(* CODESYS project TcoCore.library
   Author: Inxton
   Placeholder: TcoCore
   Title: TcoCore
   Version: 0.4.2.453
   DefaultNamespace: TcoCore
   Company: Vortex.Library

Project tree, tasks and I/O mapping:
  libraries: Tc2_EtherCAT, * (Beckhoff Automation GmbH); Tc2_Standard, 3.3.3.0 (Beckhoff Automation GmbH); Tc2_System, 3.4.24.0 (Beckhoff Automation GmbH); Tc2_Utilities, 3.3.41.0 (Beckhoff Automation GmbH); Tc3_Module, 3.3.21.0 (Beckhoff Automation GmbH)
  DUTs/
  GVLs/
  POUs/
    Compatibility/
      function block TcoContextCompatibility [ST]: _Close, _Open
      function block TcoContextNfCompatibility [ST]: Main, VolatileClose, VolatileOpen
    Prototypes/
      TcoComponent/
        interface ITcoComponent
        interface ITcoServiceable: IsService, Service
        function block TcoComponent [ST]: CheckIfIsInServiceMode, FB_init, IsService, Restore, Service, ServiceMode
      TcoContext/
        interface ITcoContext: EndCycleCount, Environment, Rtc, StartCycleCount
        interface ITcoContextEnvironment: Messaging
        function block TcoContext [ST]: Close, Context, EndCycleCount, Environment, FB_init, Identity, Main, OnEntry, OnExit, Open, Rtc, RtcSynchronize, Run, StartCycleCount
        function block TcoContextEnvironment [ST]: Messaging
      TcoMessage/
        data type eMessageCategory
        interface ITcoMessenger: Debug, Error, Info, Notify, Post, Programming, Trace, Warning
        interface ITcoMessengerSettings: IsSuspended, MinLevel, Resume, Suspend
        data type TcoMessage
        function block TcoMessenger [ST]: Catastrophic, Critical, Debug, Error, Info, Notify, Programming, Trace, Warning, Clear, Compose, FB_init, Post
        function block TcoMessengerSettings [ST]: IsSuspended, MinLevel, Resume, Suspend
      TcoObject/
        interface ITcoObject: Context, Identity
        function block TcoObject [ST]: Context, EqualsTo, FB_init, Identity, Messenger
      TcoRestorable/
        interface ITcoObjectRestorer: RestoreObject
        interface ITcoRestorable: Restore
      TcoRtc/
        interface ITcoRtc: IsSynchronized, IsValid, NowLocal, NowLocalAsTIMESTRUCT, NowUTC, NowUTCAsTIMESTRUCT, TickClock
        program RtcPrg [ST]: Synchronize
        data type RtcSynchParams
        function block TcoRtc [ST]: IsSynchronized, IsValid, NowLocal, NowLocalAsTIMESTRUCT, NowUTC, NowUTCAsTIMESTRUCT, TickClock, Update
      TcoSequencer/
        data type eSequencerError
        data type eSequencerMode
        data type eStepStatus
        interface ITcoSequencer: CurrentStep, ModeController, Run
        interface ITcoSequencerModeController: Mode, StepBackward, StepForward, StepIn
        data type StepDetails
        function block TcoSequencer [ST]: CheckStepId, Close, CompleteSequence, CompleteStep, CurrentStep, FB_init, IsStepIdUnique, Main, ModeController, OnlineChange, OnSequenceCompleted, OnSequencerError, OnStepCompleted, Open, RequestStep, Restore, Run, Step, StepChanged, StepCompleteWhen, StepInternal
        function block TcoSequencerModeController [ST]: ChangeMode, DisableModeChanging, DisableStepSkipping, Mode, OnModeChange, StepBackward, StepForward, StepIn
      TcoState/
        data type eRestoreMode
        interface ITcoState: IsAutoRestoreEnabled, LastStateChangeCycle, RestoreObject, State
        function block TcoState [ST]: ChangeState
        function block TcoStateBase [ST]: AutoRestorable, AutoRestore, ChangeStateProtected, CheckIfAutoRestoreEnabledByParent, CheckIfCalledCyclically, Context, FB_init, Identity, IsAutoRestoreEnabled, LastStateChangeCycle, OnStateChange, Restore, RestoreObject, State
        function block TcoStateExtendible [ST]: ChangeState
      TcoTask/
        data type eTaskState
        interface ITcoTask: Abort, Busy, Done, Error, Invoke
        interface ITcoTaskStatus: Busy, Done, Error
        function block TcoTask [ST]: Abort, AutoRestorable, AutoRestore, Busy, CheckIfAutoRestoreEnabledByParent, CheckIfCalledCyclically, Context, Done, DoneWhen, ElapsedTime, Enabled, Error, Execute, FB_init, Identity, Invoke, OnAbort, OnDone, OnTaskError, Ready, Restore, State, ThrowWhen
    TestFixtures/
      function block _internals_TcoContext [ST]: _Close, _GetSynchParams, _Open, _rtcUpdate, ProbeRun
      function block _internals_TcoSequencer [ST]: _Close, _Open
    Utilities/
      function block StringBuilder [ST]: Append, Clear, ToString
    program MAIN [ST]
*)

// POUs/Prototypes/TcoMessage/eMessageCategory
(*~
	<docu>
		<summary>
			Message categories.
		</summary>
	</docu>	
~*)

// ATTENTION: Values must be multiply of 100
{attribute 'qualified_only'}
{attribute 'strict'}
TYPE eMessageCategory :
(		
	All := 0,
	(*~
	<docu>
		<summary>
			Debug message to be used for debugging purpose only.
			Use when you need to report debug information for you as programmer. 
		</summary>
	</docu>	
	~*)	
	Debug := 100,
	(*~
	<docu>
		<summary>
			Trace message to be used for tracing purpose.
			Use when you need to track detailed information about internal states of the program for detailed visibility. 
			This is lowest level of category that can be used in production, for detailed observation of PLC program.
		</summary>
	</docu>	
	~*)	
	Trace := 200,
	(*~
	<docu>
		<summary>
			Info message.
			Use when you want to deliver information to the user, that has only informative character and does not adversely affect a process.
		</summary>
	</docu>	
	~*)	
	Info := 300,
	(*~
	<docu>
		<summary>
			Time-out message.
			Use this category when you want to report a timed-out information, that may eventually succed.
		</summary>
	</docu>	
	~*)
	TimedOut := 400,
	(*~
	<docu>
		<summary>
			Notification message.
			Use this category when you want to report a notification that may be of interest to the user, but does not adversly affect a process.
		</summary>
	</docu>	
	~*)
	Notification := 500,
	(*~
	<docu>
		<summary>
			Warning message.
			Use this category when you want to report to the user an information about a possible problem, that may adversly affect a process.
			Information in this cateogory aims to help the user to identify a problem, the cause of such problem does not necessarily stops the process.
		</summary>
	</docu>	
	~*)
	Warning := 600,
	(*~
	<docu>
		<summary>
			Error message.
			Use this categoty when there is a failure that cannot be immediately recovered and an intervention is needed. This is typically a situation when a device fails
			to deliver expected result. 
			Do not use this category to report information about failed process like measurement or detection.
		</summary>
	</docu>	
	~*)
	Error := 700,	
	(*~
	<docu>
		<summary>
			Programming issue.
			Use this category to inform about a possible programming error, defect in settings or missing information at a level of programming or system or process settings. 
		</summary>
	</docu>	
	~*)
	ProgrammingError := 900,
	(*~
	<docu>
		<summary>
			Critical error. 
			Use this category when a critical error occured, that is not recoverable by the means of software (reset/restore) and a detailed inspection is required.
		</summary>
	</docu>	
	~*)	
	Critical := 1000,		
	(*~
	<docu>
		<summary>
			Catastrophic error. 
			Use this category when there is a situation when the device cannot continue operations due to irrecoverable failure.
		</summary>
	</docu>	
	~*)
	Catastrophic := 1100,
	
	None := 32767
);
END_TYPE

// POUs/Prototypes/TcoMessage/TcoMessage
(*~
	<docu>
		<summary>
			Complete message details including time stamp, message text, message category, identity of the message provider, context cycle in which the message was posted.			
		</summary>				
	</docu>	
~*)
TYPE TcoMessage :
STRUCT
(*~
	<docu>
		<summary>
			Time when the message was posted.
		</summary>				
	</docu>	
~*)
	{attribute clr [ReadOnly()]}
	TimeStamp : DT;
(*~
	<docu>
		<summary>
			Text of the message.
		</summary>				
	</docu>	
~*)
	{attribute clr [ReadOnly()]}		
	Text : STRING(125);
(*~
	<docu>
		<summary>
			Identity of the TcoObject that posted this message. 
		</summary>				
	</docu>	
~*)
	{attribute clr [ReadOnly()]}	
	Identity : ULINT;	
(*~
	<docu>
		<summary>
			Message category of this message. See <see cref="eMessageCategory"/> for detailed informations. 
		</summary>				
	</docu>	
~*)
	Category : eMessageCategory;
(*~
	<docu>
		<summary>
			Context cycle in which the message was posted.
		</summary>				
	</docu>	
~*)
	{attribute clr [ReadOnly()]}
	Cycle : ULINT;
	
(*~
	<docu>
		<summary>
			Count of messages of the object in the current cycle.
		</summary>				
	</docu>	
~*)
	{attribute clr [ReadOnly()]}
	PerCycleCount : BYTE;
END_STRUCT
END_TYPE

// POUs/Prototypes/TcoRtc/RtcSynchParams
TYPE RtcSynchParams :
STRUCT
	synchContextIdentity	:	ULINT;
	doSynch					:	BOOL;
	syncAmsId				:	STRING;
	syncPeriod				:	UINT; 
END_STRUCT
END_TYPE

// POUs/Prototypes/TcoSequencer/eSequencerError
(*~
	<docu>
		<summary>
			Describes cause of the sequencer error.
		</summary>				
	</docu>	
~*)
{attribute 'qualified_only'}
{attribute 'strict'}
TYPE eSequencerError :
(
(*~
	<docu>
		<summary>
			No error.
		</summary>				
	</docu>	
~*)	
	noError := 0,
(*~
	<docu>
		<summary>
			Some of the StepId in the sequence is not unique (```TcoSequencer.Step(StepID)```).
		</summary>				
	</docu>	
~*)	
	NotUniqueStepId := 10,
(*~
	<docu>
		<summary>
			StepId of the currently executed step has been changed during execution.
		</summary>				
	</docu>	
~*)
	StepIdHasBeenChanged := 20,
(*~
	<docu>
		<summary>
			Order of the currently executed step has been changed during execution.
		</summary>				
	</docu>	
~*)
	OrderOfTheStepHasBeenChanged := 40,
(*~
	<docu>
		<summary>
			Method ```RequestStep``` has been called with nonexisting StepId.
		</summary>				
	</docu>	
~*)
	StepWithRequestedIdDoesNotExists := 50,
(*~
	<docu>
		<summary>
			Multiple simultaneous calls of ```RequestStep()```. Another ```RequestStep()``` method has been called while previous ```RequestStep()``` call has not yet been completed.
		</summary>				
	</docu>	
~*)
	MultipleRequestStepMethodCall := 60,
(*~
	<docu>
		<summary>
			StepId is bellow min. range. Minimal value is -32767.
		</summary>				
	</docu>	
~*)
	StepIdTooLow := 70,
(*~
	<docu>
		<summary>
			StepId is above max range. Maximal value is 32766.
		</summary>				
	</docu>	
~*)
	StepIdTooHigh := 80,
(*~
	<docu>
		<summary>
			Mode of the sequencer is invalid.
		</summary>				
	</docu>	
~*)
	InvalidSequencerMode := 90
);
END_TYPE

// POUs/Prototypes/TcoSequencer/eSequencerMode
(*~
	<docu>
		<summary>
			Modes of the sequencer.
		</summary>				
	</docu>	
~*)	
{attribute 'qualified_only'}
{attribute 'strict'}
TYPE eSequencerMode :
(
(*~
	<docu>
		<summary>
			Invalid, no logic is executed.
		</summary>				
	</docu>	
~*)	
	Invalid := -10,
(*~
	<docu>
		<summary>
			Sequencer runs the steps of the sequence. 
			(When cyclic mode is selected, next step is automatically started after the previous one has been completed.)
		</summary>				
	</docu>	
~*)	
	CyclicMode := 0,
(*~
	<docu>
		<summary>
		    Sequencer is in mode of step-by-step operation. The current step completes the execution regularly.
			In this mode the Step Forward/Backward and manual step execution is available.			
			<para>
				See <see cref="TcoSequencerModeController.PlcTcoSequencerModeController.StepForward()"/> for detailed description.
				See <see cref="TcoSequencerModeController.PlcTcoSequencerModeController.StepIn()"/> for detailed description.
				See <see cref="TcoSequencerModeController.PlcTcoSequencerModeController.StepBackward()"/> for detailed description.
			</para>
		</summary>				
	</docu>	
~*)	
	StepMode := 10
);
END_TYPE

// POUs/Prototypes/TcoSequencer/eStepStatus
(*~
	<docu>
		<summary>
			Describes the step status inside the sequencer.
		</summary>				
	</docu>	
~*)
{attribute 'qualified_only'}
{attribute 'strict'}
TYPE eStepStatus :
(
(*~
	<docu>
		<summary>
			No status defined.
		</summary>				
	</docu>	
~*)	
	None := 0,
(*~
	<docu>
		<summary>
			Step is disabled and won't be executed.
			Next enabled step in the sequence will be executed, when the sequencer reaches that step.
		</summary>				
	</docu>	
~*)	
	Disabled := 10,
(*~
	<docu>
		<summary>
			Step is ready to run. This case occurs when sequence is in step mode, step is in order of the execution and step is enabled.
			The body statements of the current step's are not executing. After calling StepIn method, step starts running the statements.
		</summary>				
	</docu>	
~*)	
	ReadyToRun := 20,
(*~
	<docu>
		<summary>
			Step is currently running (The body statements are running).
		</summary>				
	</docu>	
~*)	
	Running := 30,	
(*~
	<docu>
		<summary>
			Step has finished (The body statements are not running).
		</summary>				
	</docu>	
~*)	
	Done := 40,
(*~
	<docu>
		<summary>
			Step is in error state. The sequencer does not execute any step logic.
		</summary>				
	</docu>	
~*)	
	Error := 50
);
END_TYPE

// POUs/Prototypes/TcoSequencer/StepDetails
(*~
	<docu>
		<summary>
			Describes the status of a step of the sequencer.
		</summary>				
	</docu>	
~*)
TYPE StepDetails :
STRUCT
(*~
	<docu>
		<summary>
			Step identification number.
		</summary>	
		<remarks>			
 			<note type="important">
				This number must be unique throughout the complete sequence. It is required to uniquely identify the step of the sequence.
			</note>
			<para>
				The <see cref="TcoSequencer.PlcTcoSequencer.RequestStep"/> method is using this number to jump to the required step.
			</para>
		</remarks>
	</docu>	
~*)
	{attribute addProperty Name "<#Step ID#>"}
	ID: INT;
(*~
	<docu>
		<summary>
			Order of the step in the sequence.
		</summary>	
	</docu>	
~*)
	{attribute addProperty Name "<#Step Order#>"}
	Order: UINT;
(*~
	<docu>
		<summary>
			If this value is false, step body is not executed and execution is moved to the next enabled step in the sequence.
		</summary>				
	</docu>	
~*)
	{attribute addProperty Name "<#Enabled#>"}
	Enabled: BOOL;
(*~
	<docu>
		<summary>
			Step description text.
		</summary>				
	</docu>	
~*)
	{attribute addProperty Name "<#Step description#>"}
	Description: STRING(254);
(*~
	<docu>
		<summary>
			Describes step status.
		</summary>				
		<remarks>			
			<para>
				See <see cref="eStepStatus"/> for detailed description.
			</para>
		</remarks>		
		enumStepStatus
	</docu>	
~*)	
	{attribute addProperty Name "<#Step status#>"}
	Status : eStepStatus;
(*~
	<docu>
		<summary>
			Step duration time.
		</summary>				
	</docu>	
~*)	
	{attribute addProperty Name "<#Step duration#>"}
	Duration : TIME;
END_STRUCT
END_TYPE

// POUs/Prototypes/TcoState/eRestoreMode
{attribute 'qualified_only'}
{attribute 'strict'}
TYPE eRestoreMode :
(
	None := 0,
	
	(*~
	<docu>
		<summary>
				Activates automatic restore mechanism for all immediate children (direct members).
		</summary>				
	</docu>	
	~*)	
	AutoRestoreMembers := 10
);
END_TYPE

// POUs/Prototypes/TcoTask/eTaskState
(*~
	<docu>
		<summary>
			Describes the state of the respective task.
		</summary>				
	</docu>	
~*)
{attribute 'qualified_only'}
{attribute 'strict'}
TYPE eTaskState :
(
(*~
	<docu>
		<summary>
			Task is in Ready state, the Execute() method returns FALSE. 
			Task can be started by calling the Invoke() method. 
		</summary>				
	</docu>	
~*)
	Ready := 0,
(*~
	<docu>
		<summary>
			Task is in Requested state, if Invoke() method has been called and the Execute() method has not been called yet. The first following call of the method Execute() 
			change the task state to Executing and returns TRUE, until Done or Error state is reached.
		</summary>				
	</docu>	
~*)
	Requested := 10,
(*~
	<docu>
		<summary>
			When the task is in Busy state, Execute() method returns TRUE. Leaving this state is possible as follows:
			<para>1.) By calling the Abort() task gets into the Idle state.</para>
			<para>2.) By calling the DoneWhen(true) task gets into the Done state.</para>
			<para>3.) By calling the Restore() task gets into the Idle state.</para>
			<para>4.) By calling the ThrowWhen(true) task gets into the Error state.</para>
		</summary>				
	</docu>	
~*)
	Busy := 20,
(*~
	<docu>
		<summary>
			Task is in Error state. To be able to start the task again the error state has to be reseted by calling the Restore() method.
		</summary>				
	</docu>	
~*)	
	Error := 30,
(*~
	<docu>
		<summary>
			Task is in Done state, Execute() method returns FALSE. To be able to start the task again '''rising edge''' of the calling of the Invoke() method needs to be performed.
			<p>Analogously to the xExecute signal of the <a href="https://plcopen.org/sites/default/files/downloads/creating_plcopen_compliant_function_block_libraries.pdf" title="Title"> PLCopen </a> motion function blocks.</p>
		</summary>				
	</docu>	
~*)	
	Done := 40
);
END_TYPE

// POUs/Compatibility/TcoContextCompatibility
{attribute 'hide'}
{attribute clr [ExcludeFromApiDocumentation()]}
FUNCTION_BLOCK ABSTRACT TcoContextCompatibility EXTENDS TcoContext

{attribute 'hide'}
METHOD PROTECTED FINAL _Close
THIS^.Close();
END_METHOD

{attribute 'hide'}
METHOD PROTECTED FINAL _Open
THIS^.Open();
END_METHOD

END_FUNCTION_BLOCK

// POUs/Prototypes/TcoContext/TcoContext

(*~
	<docu>
		<summary>
			Root construction container, provides context information for <c>TcoObjects</c> declared within its scope.
			This function block is ```abstract``` and cannot be instantiated. 
			Use <see cref="TcoContext.PlcTcoContext.Run()"/> to run this context, ```Run``` method must be called only once per PLC Task cycle.
			Several 'TcoContext' instances can be declared and called inside one TwinCAT PlcTask, but only once per PLC cycle. 
			The instance should not be accessed from several Twincat PlcTasks.
			Default implemenation of the 'TcoContext' allows its child members access properties <see cref="TcoContext.PlcTcoContext.StartCycleCount()"/> 
			and <see cref="TcoContext.PlcTcoContext.EndCycleCount()"/>, messenger settings, rtc and other information related to the context of the running logic.			 			 			
			<note type="tip">
				 A <c>TcoContext</c> can contain objects, components and PLC logic of one independent station of the machine, 
				 while the another one can cover the same for another station.			
			</note>
			<remarks>			
				<note type="tip">
					TwinCAT PlcTask and <see cref="TcoTask.PlcTcoTask()"/> refer to two different concepts. 
				</note>
			</remarks>
		</summary>	
		<example>
			Declaration part of the 'TcoContext' example. 
		</example>
		<example>
				[!code-pas[Main](~/../TcOpen/src/TcoApplicationExamples/XaeAppExamples/PlcAppExamples/POUs/Context/VitoCorleone_Context.TcPOU?name=ContextExampleDeclarations)]
		</example>
		<example>
			Implementation part of the 'TcoContext' example.
		</example>
		<example>
				[!code-pas[Main](~/../TcOpen/src/TcoApplicationExamples/XaeAppExamples/PlcAppExamples/POUs/Context/VitoCorleone_Context.TcPOU?name=ContextExampleCode)]
		</example>
	</docu>	
~*)
FUNCTION_BLOCK PUBLIC ABSTRACT TcoContext IMPLEMENTS ITcoContext
VAR
	(*~
		<docu>
			<summary>
				Identity of this <c>TcoContext</c>.
				This variable is used in the higher level applications, 
				it allows to identify the context in SCADA like applications.	  
			</summary>			
		</docu>	
	~*)
	{attribute clr [RenderIgnore()]}
	{attribute clr [ReadOnly()]}
	_Identity : ULINT;
	{attribute clr [ReadOnly()]}
	_startCycleCount : ULINT;
	{attribute clr [ReadOnly()]}
	_endCycleCount : ULINT;
	_messagingLevel : eMessageCategory;
	{attribute clr [ReadOnly()]}
	_rtc : TcoRtc;
	{attribute clr [RenderIgnore()]}
    _settings : TcoContextEnvironment;	
END_VAR

(*~
	<docu>
		<summary>
			This method is called implicitly at the entry point of this context (<see cref="TcoContext.PlcTcoContext.Run()"/>).
			<remarks>			
				<note type="important">
					Do not call this method explicitly!
				</note>
			</remarks>
		</summary>			
	</docu>	
~*)
METHOD INTERNAL FINAL Close
_endCycleCount := _startCycleCount;
END_METHOD

(*~
	<docu>
		<summary>
			Returns reference to this instance of the <see cref="TcoContext.PlcTcoContext()"/>.
		</summary>			
	</docu>	
~*)
PROPERTY Context : ITcoContext
GET
Context := THIS^;
END_GET
END_PROPERTY

(*~
	<docu>
		<summary>
		    Gets the value of the counter incrememented by '1' at the end of each execution of this <see cref="TcoContext.PlcTcoContext()"/>.			
		</summary>			
	</docu>	
~*)
PROPERTY EndCycleCount : ULINT
GET
EndCycleCount := _endCycleCount;
END_GET
END_PROPERTY

PROPERTY Environment : ITcoContextEnvironment
GET
Environment := _settings;
END_GET
END_PROPERTY

METHOD FB_init : BOOL
VAR_INPUT
	bInitRetains : BOOL; // if TRUE, the retain variables are initialized (warm start / cold start)
	bInCopyCode : BOOL;  // if TRUE, the instance afterwards gets moved into the copy code (online change)
END_VAR
_Identity := ADR(THIS^);
END_METHOD

(*~
	<docu>
		<summary>
			Returns the identity of this <see cref ="TcoContext.PlcTcoContext()"/>. 
			This value is assigned when instantiated and cannot be changed at runtime.
			This member is used in the higher level applications.  
		</summary>			
	</docu>	
~*)
PROPERTY Identity : ULINT
GET
Identity := _Identity;
END_GET
END_PROPERTY

(*~
	<docu>
		<summary>
			Main method of the TcoContext. This is the entry point of any control logic that belongs to this context. 
			The call of this method is ensured by calling the <c>InstanceName.Run()</c> method, and it must not be called explicitly.
			This method is abstract, and it must be overridden in derived block.
		</summary>
	</docu>
~*)
METHOD PROTECTED ABSTRACT Main
END_METHOD

(*~
	<docu>
		<summary>
			Called on entry into context. When overridden in derived class allows to execute an arbitrary logic prior to opening the context cycle.
			<remarks>			
				<note type="important">					
					The method executes prior to opening the context. The context might not be properly initialized on first call. 
					Any information contained in the context at this point are from the last execution.
				</note>
			</remarks>
		</summary>			
	</docu>	
~*)
METHOD PROTECTED OnEntry
END_METHOD


(*~
	<docu>
		<summary>
			Called upon exit from the context. When overridden in derived class allows to execute an arbitrary logic after closing the context cycle.	
		</summary>			
	</docu>	
~*)METHOD PROTECTED OnExit
END_METHOD

(*~
	<docu>
		<summary>
			This method is called implicitly at the entry point of this context (<see cref="TcoContext.PlcTcoContext.Run()"/>).
			<remarks>			
				<note type="important">
					Do not call this method explicitly.
				</note>
			</remarks>
		</summary>			
	</docu>	
~*)
METHOD INTERNAL FINAL Open
_startCycleCount := _startCycleCount + 1;
_rtc.Update();
END_METHOD

PROPERTY Rtc : ITcoRtc
GET
Rtc := _rtc;
END_GET
END_PROPERTY

(*~
	<docu>
		<summary>
			Syncronizes the Real Time Clock (RTC) from given source.
			<remarks>			
				<note type="important">
					There is single RTC source for entire application. All context share the same RTC source.
				</note>
			</remarks>
		</summary>			
	</docu>	
~*)
METHOD RtcSynchronize  : REFERENCE TO TcoContext
VAR_INPUT
	(*~
		<docu>
			<summary>
				When called with true the synchronization mechanism executes.		
			</summary>			
		</docu>	
	~*)
	inDoSynch				:	BOOL;
	(*~
		<docu>
			<summary>
				```AMS ID``` of the system against which RTC of this application will synchronize.			
			</summary>			
		</docu>	
	~*)
	inSyncAmsId				:	STRING;
	(*~
		<docu>
			<summary>
				Set the synchronisation period.		
			</summary>			
		</docu>	
	~*)
	inSyncPeriod			:	UINT; 
END_VAR

VAR
	_RtcSynchParams			:	RtcSynchParams;			
END_VAR
_RtcSynchParams.doSynch					:=	inDoSynch;
_RtcSynchParams.syncAmsId				:=	inSyncAmsId;
_RtcSynchParams.syncPeriod				:=	inSyncPeriod;
_RtcSynchParams.synchContextIdentity	:=	THIS^._Identity;
RtcPrg.Synchronize(_RtcSynchParams);
RtcSynchronize REF= THIS^;
END_METHOD

(*~
	<docu>
		<summary>
			<para>
				This method executes of this context. It provided correct order of execution order of inner methods. Any logic of this context must be called within <see cref="TcoContext.PlcTcoContext.Main()"/>
				method. This method is final, so it cannot be overriden. The <c>InstanceName.Run()</c> needs to be called cyclically.
			</para>
		</summary>			
	</docu>	
~*)
METHOD PUBLIC FINAL Run
THIS^.OnEntry();
THIS^.Open();
THIS^.Main();
THIS^.Close();
THIS^.OnExit();
END_METHOD

(*~
	<docu>
		<summary>
		    Gets number of executions of this context. Value of this property is incremented by '1' at the beginning of the <see cref="TcoContext.PlcTcoContext()"/>. 			 			
		</summary>			
	</docu>	
~*)
PROPERTY StartCycleCount : ULINT
GET
StartCycleCount := _startCycleCount;
END_GET
END_PROPERTY

END_FUNCTION_BLOCK

// POUs/Prototypes/TcoTask/TcoTask
(*~
	<docu>
		<summary>
			Provides basic task execution. Task could be started by calling the <see cref="TcoTask.PlcTcoTask.Invoke()"/> method. The  <see cref="TcoTask.PlcTcoTask.Execute()"/> method returns true, until the task reaches the Done state.
			<para>
				To get the actual state of the task, <see cref="TcoTask.PlcTcoTask.Ready()"/>, <see cref="TcoTask.PlcTcoTask.Busy()"/>, <see cref="TcoTask.PlcTcoTask.Error()"/> and <see cref="TcoTask.PlcTcoTask.Done()"/> properties are available.
			</para>
		</summary>
		<example>
			Declaration part of the 'TcoTask' example. 
		</example>
		<example>
			[!code-pas[Main](~/../TcOpen/src/TcoApplicationExamples/XaeAppExamples/PlcAppExamples/POUs/Task/AskForTheFavor_Task.TcPOU?name=TaskExampleDeclarations)]
		</example>
		<example>
			Implementation part of the 'TcoTask' example.
		</example>
		<example>
			[!code-pas[Main](~/../TcOpen/src/TcoApplicationExamples/XaeAppExamples/PlcAppExamples/POUs/Task/AskForTheFavor_Task.TcPOU?name=TaskBodyExampleCode)]
		</example>
		<example>
			Example of the invoking this example 'TcoTask' instance 'outside' of the instance and wait if it ends-up in 'DONE' state or in 'ERROR' state.
		</example>
		<example>
			[!code-pas[Main](~/../TcOpen/src/TcoApplicationExamples/XaeAppExamples/PlcAppExamples/POUs/Sequencer/MakeAnOfferThatCantBeRefused.TcPOU?name=TaskExternalUseExample)]
		</example>
	</docu>	
~*)	
FUNCTION_BLOCK TcoTask EXTENDS TcoObject IMPLEMENTS ITcoTask, ITcoTaskStatus
VAR
	{attribute clr [ReadOnly()]}
	_taskState : eTaskState;
	{attribute 'hide'}
	_nextExpectedCycle : ULINT;
	{attribute 'hide'}
	_AutoRestorable : BOOL;
	{attribute 'hide'}
	_StartCycleCount	: ULINT;
	{attribute 'hide'}
	_MyParentsChangeStateCycle	: ULINT;
	{attribute 'hide'}
	_MyParentsLastChangeState	: INT;	
(*~
	<docu>
		<summary>
			Use to restore this instance to the Ready state. The value is than set to FALSE.			
		</summary>		
	</docu>	
~*)	
	{attribute addProperty Name "<#Restore request#>"}
	_restoreRequest : BOOL;
(*~
	<docu>
		<summary>
			Use to start the execution of the task from Ready state or from Done state by performing the rising edge. 
			<p>Analogously to the xExecute signal of the <a href="https://plcopen.org/sites/default/files/downloads/creating_plcopen_compliant_function_block_libraries.pdf" title="Title"> PLCopen </a> motion function blocks.</p>			
		</summary>			
	</docu>	
~*)
	{attribute addProperty Name "<#Invoke request#>"}
	_invokeRequest : BOOL;
(*~
	<docu>
		<summary>
			Use to abort the executing task and set this instance back to the Ready state.
			The value is than set to FALSE. 
		</summary>			
	</docu>	
~*)
	{attribute addProperty Name "<#Abort request#>"}
	_abortRequest : BOOL;	
(*~
	<docu>
		<summary>
			Use to determine if the task execution is enabled for example from the HMI application. 
			This value is read only, to modify it use the property <see cref="TcoTask.PlcTcoTask.Enabled()"/>		
		</summary>		
	</docu>	
~*)	
	{attribute addProperty Name "<#Enabled#>"}
	{attribute clr [ReadOnly()]}
	_enabled : BOOL := TRUE;
END_VAR

VAR	
	{attribute 'hide'}
	_executionTimer : Tc2_Standard.TON;
	{attribute clr [ReadOnly()]}
	_elapsedTime : TIME;
END_VAR

(*~
	<docu>
		<summary>
			Aborts the execution of this task and restores the ready state.			
		</summary>			
	</docu>	
~*)
METHOD Abort
IF THIS^._taskState = eTaskState.Busy THEN
	OnAbort();
	THIS^.Restore();
END_IF
END_METHOD

(*~
	<docu>
		<summary>
			Gets whether this instance is auto restorable. This is depends on the parent's settings; the value of this property is given by the parent of this object. 
			This value is assigned after download by calling the implicit method <c>FB_init()</c> of the parent object and cannot be changed during runtime.
			The <c>AutoRestorable</c> property of this objects is retrieved from the <c>EnableAutoRestore</c> property of the parent object.
			This is done by calling the <c>CheckIfAutoRestoreEnabledByParent()</c> method inside the implicit method <c>FB_init()</c> after download.
			If this instance is the auto restorable it will call the <see cref="TcoTask.PlcTcoTask.Restore()"/> method if:
			<para>
				1.) The <see cref="TcoTask.PlcTcoTask.Invoke()"/> method has not been called for one or more cycles and starts to be called again.
			</para>
			<para>
				2.)	Parent object of this instance changes its state.
			</para>
			<para>
				See also <see cref="TcoTask.PlcTcoTask.EnableAutoRestore()"/>
			</para>
		</summary>			
	</docu>	
~*)
PROPERTY AutoRestorable : BOOL
GET
AutoRestorable := _AutoRestorable;
END_GET
END_PROPERTY

(*~
	<docu>
		<summary>
			Private method called each time that the <see cref="TcoTask.PlcTcoTask.Execute()"/> method is called. If this instance is auto restorable, this method ensures calling the <see cref="TcoTask.PlcTcoTask.Restore()"/> method if:
			<para>
				1.)	Parent object of this instance changes its state in this Plc cycle.
			</para>
			<para>
				2.)	Parent object of this instance changes its state no mather when and this instance has not yet process this change.
			</para>
			<para>
				3.) The <see cref="TcoTask.PlcTcoTask.Invoke()"/> method has not been called for one or more cycles and starts to be called again.
			</para>
			<para>
				See also <see cref="TcoTask.PlcTcoTask.AutoRestorable()"/>
			</para>
			<para>
				See also <see cref="TcoTask.PlcTcoTask.EnableAutoRestore()"/>
			</para>
		</summary>			
	</docu>	
~*)
METHOD PRIVATE AutoRestore
VAR 
	_MyParent_TcoState	: ITcoState := 0;
	_MyParent_ChangeStateCycle : ULINT;
	_MyParent_LastChangeState : INT;
END_VAR
// If the parent of this instance is TcoState type or its derived type and the parent
// EnableAutoRestore property is set to TRUE, this instance determines the value
// of its own AutoRestorable property by calling CheckIfAutoRestoreEnabledByParent 
// after each download.
IF _AutoRestorable THEN		
	IF __QUERYINTERFACE(THIS^._Parent,_MyParent_TcoState) THEN 
		_MyParent_ChangeStateCycle := _MyParent_TcoState.LastStateChangeCycle;
		_MyParent_LastChangeState := _MyParent_TcoState.State;
	END_IF;	
	//If OnStateChange event of the parent has occured, the value of the parent's 
	//StartCycleCount property is stored into its ChangeStateCycle property.
	//Each child has to deal with it individually in the next call of its body,
	//restore itself, and copy the parent's ChangeStateCycle property into the
	//child's own property.
	IF _MyParent_ChangeStateCycle <> _MyParentsChangeStateCycle THEN
		Restore();
		_MyParentsChangeStateCycle := _MyParent_ChangeStateCycle;
	END_IF
	IF _MyParent_LastChangeState <> _MyParentsLastChangeState THEN
		Restore();
		_MyParentsLastChangeState := _MyParent_LastChangeState;
	END_IF
END_IF
END_METHOD

(*~
	<docu>
		<summary>
			Gets whether the task is executing.
		</summary>			
	</docu>	
~*)
PROPERTY Busy : BOOL
GET
Busy := THIS^._taskState = eTaskState.Busy;
END_GET
END_PROPERTY

(*~
	<docu>
		<summary>
			This method ensures reading out the parent's <see cref="TcoState.PlcTcoState.EnableAutoRestore()/> property and writing it into the <see cref="TcoTask.PlcTcoTask.AutoRestorable()"/> of this instance.
			Calling this method is ensured by calling the implicit method <c>FB_init()</c> after download, or after online change.
		</summary>			
	</docu>	
~*)
{attribute 'call_after_online_change_slot' := '100'}
METHOD PRIVATE CheckIfAutoRestoreEnabledByParent
VAR
	_MyParent_TcoState	: 	ITcoState := 0;
END_VAR
IF __QUERYINTERFACE(THIS^._Parent,_MyParent_TcoState) THEN 
	_AutoRestorable := _MyParent_TcoState.IsAutoRestoreEnabled;
END_IF;
END_METHOD

(*~
	<docu>
		<summary>
			Private method called inside the <see cref="TcoTask.PlcTcoTask.Execute()"/> method checking the cyclicall calling of this method. 
			If this instance is auto restorable, this method ensures calling the <see cref="TcoTask.PlcTcoTask.Restore()"/> method if
			the <see cref="TcoTask.PlcTcoTask.Execute()"/> method has not been called for one or more cycles and starts to be called again.
			<para>
				See also <see cref="TcoTask.PlcTcoTask.AutoRestorable()"/>
			</para>
			<para>
				See also <see cref="TcoTask.PlcTcoTask.EnableAutoRestore()"/>
			</para>
		</summary>			
	</docu>	
~*)
{attribute clr [ExcludeFromApiDocumentation()]}
METHOD PRIVATE CheckIfCalledCyclically
VAR 
	_MyContextStartCycleCount : ULINT;
END_VAR
//If parent of this instance is TcoState type or its derived type and the parent
//EnableAutoRestore property is set to TRUE, this instance determines the value
//of its own AutoRestorable property by calling CheckIfAutoRestoreEnabledByParent 
//after each download.
IF _AutoRestorable THEN		
	_MyContextStartCycleCount := THIS^.Context.StartCycleCount;
	//If this instance is AutoRestorable, its body has to be called cyclically, 
	//otherwise this instance is restored.
	//This mechanism force the user to call this instance properly,
	//in order to don't miss the OnStateChange() event of the parent
	//in case of the body of this instance isn't called.
	IF _MyContextStartCycleCount > _StartCycleCount + 1 THEN
		Restore();
	END_IF
	_StartCycleCount := _MyContextStartCycleCount;
END_IF
END_METHOD

(*~
	<docu>
		<summary>
			Gets the context of this object.
			This context is given by declaration, its value is assigned after download by calling the implicit method <c>FB_init()</c> and cannot be changed during runtime.
		</summary>			
	</docu>	
~*)
PROPERTY Context : ITcoContext
GET
Context := THIS^._Parent.Context;
END_GET
END_PROPERTY

(*~
	<docu>
		<summary>
			Gets whether the task has succesfully completed the  execution and did not enter into the Error state.
		</summary>			
	</docu>	
~*)
PROPERTY Done : BOOL
GET
Done := THIS^._taskState = eTaskState.Done;
END_GET
END_PROPERTY

(*~
	<docu>
		<summary>
			Completes the execution of this task when ```inCondition``` is true; the task transitions into ```Done``` state.
		</summary>			
	</docu>	
~*)
METHOD DoneWhen 
VAR_INPUT
	inCondition : BOOL;
END_VAR
IF (inCondition) THEN
	THIS^._taskState := eTaskState.Done;
	OnDone();			
END_IF;
END_METHOD

(*~
	<docu>
		<summary>
			Gets the elapsed time of the execution of this task. 
			<remarks>			
				<note type="important">
					Uses `TIME` type. It might be not sutable for tasks running longer than 49 days.
				</note>
			</remarks>		
		</summary>			
	</docu>	
~*)
PROPERTY PUBLIC ElapsedTime : TIME
GET
ElapsedTime := _elapsedTime;
END_GET
END_PROPERTY

(*~
	<docu>
		<summary>
			Gets whether the task execution is enabled.
			The task can start with <see cref="TcoTask.PlcTcoTask.Invoke()"/> method call only when this property si TRUE. 
			If the task is ```Busy``` and this property transitions to ```FALSE```, the task stops execution and enters ```Error``` state. 
		</summary>			
	</docu>	
~*)
PROPERTY Enabled : BOOL
GET
Enabled := _enabled;
END_GET
SET
_enabled := Enabled;
END_SET
END_PROPERTY

(*~
	<docu>
		<summary>
			Returns true if the task has is in error state. To be able to start the the task again, <see cref="TcoTask.PlcTcoTask.Restore()"/> method needs to be called before 
			restarting it again calling <see cref="TcoTask.PlcTcoTask.Invoke()"/> method.
		</summary>			
	</docu>	
~*)
PROPERTY Error : BOOL
GET
Error := THIS^._taskState = eTaskState.Error;
END_GET
END_PROPERTY

(*~
	<docu>
		<summary>
			Returns true if the task is Busy, otherwise false.
			This method needs to be called cyclically.
		</summary>			
	</docu>	
~*)
METHOD Execute : BOOL
VAR
	_serviceableParent : ITcoServiceable;
END_VAR

VAR
	tmpTimeDiff : TIME;
END_VAR
// Detects if parent is in serviceable state to enable manual invoke of the task from the HMI/SCADA system.
IF(THIS^._Parent <> 0 )THEN
	IF(__QUERYINTERFACE(THIS^._Parent, _serviceableParent)) THEN
		IF(NOT _serviceableParent.IsService) THEN
			THIS^._invokeRequest := FALSE;
		END_IF
	END_IF
END_IF;

//Triggering Invoke from remote system
IF(THIS^._taskState = eTaskState.Ready AND THIS^._invokeRequest) THEN
	THIS^.Invoke();
END_IF;
THIS^._invokeRequest := FALSE;

//Triggering Abort from remote system
IF((THIS^._taskState = eTaskState.Requested OR THIS^._taskState = eTaskState.Busy) AND THIS^._abortRequest) THEN
	THIS^.Abort();
	THIS^._abortRequest := FALSE;
END_IF;

//Triggering Restore from remote system
IF( THIS^._restoreRequest) THEN
	THIS^.Restore();
	THIS^._restoreRequest := FALSE;
END_IF;

IF NOT _enabled THEN
	IF THIS^._taskState = eTaskState.Requested THEN		
		THIS^.Messenger.Post('Task cannot start; Enabled property is FALSE.',eMessageCategory.Info);	
		THIS^.Restore();
	END_IF
	IF THIS^._taskState = eTaskState.Busy THEN
		THIS^.Messenger.Post('Running task entered Error state since the Enabled property transitioned to FALSE during task execution.',eMessageCategory.Error);	
		THIS^._taskState := eTaskState.Error;
	END_IF
END_IF;

CheckIfCalledCyclically();
AutoRestore();

IF(THIS^._taskState = eTaskState.Requested) THEN	
	_executionTimer(IN := FALSE);
	THIS^._taskState := eTaskState.Busy;
END_IF;

IF(THIS^._taskState = eTaskState.Error) THEN
	OnTaskError();
END_IF;
	
Execute := (THIS^._taskState = eTaskState.Busy);

IF(Execute) THEN
	_executionTimer(IN := Execute, PT := T#49D);
	_elapsedTime := _executionTimer.ET;
END_IF;
END_METHOD

METHOD PUBLIC FB_init : BOOL
VAR_INPUT
	bInitRetains : BOOL; // if TRUE, the retain variables are initialized (warm start / cold start)
	bInCopyCode : BOOL;  // if TRUE, the instance afterwards gets moved into the copy code (online change)
	Parent : ITcoObject;
END_VAR
_Parent := Parent;

CheckIfAutoRestoreEnabledByParent();
END_METHOD

(*~
	<docu>
		<summary>
			Gets identity of this <see cref ="TcoTask.PlcTcoTask()"/>. 
			This value is assigned after download by calling the implicit method <c>FB_init()</c> and cannot be changed during runtime.
			This variable is used in the higher level applications.  
		</summary>			
	</docu>	
~*)
PROPERTY Identity : ULINT
GET
Identity := _Identity;
END_GET
END_PROPERTY

(*~
	<docu>
		<summary>
			Use to start the execution of the task. The starting is possible from Ready state.
			<para>Moreover it is also possible to start the task again from Done state by performing the '''rising edge''' of the calling of the Invoke() method.</para>
			<p>Analogously to the xExecute signal of the <a href="https://plcopen.org/sites/default/files/downloads/creating_plcopen_compliant_function_block_libraries.pdf" title="Title"> PLCopen </a> motion function blocks.</p>			
		</summary>			
	</docu>	
~*)
METHOD Invoke : ITcoTaskStatus
VAR
	_newInvokeCall	:	BOOL;
END_VAR
_newInvokeCall := THIS^._Parent.Context.StartCycleCount > _nextExpectedCycle;

IF(THIS^._taskState = eTaskState.Ready OR (THIS^._taskState = eTaskState.Done AND _newInvokeCall)) THEN
	IF _enabled THEN
		THIS^._taskState := eTaskState.Requested;
	ELSE
		THIS^.Messenger.Post('Task cannot be started  as its Enabled property is FALSE.',eMessageCategory.Info);
	END_IF	
END_IF	

_nextExpectedCycle := THIS^._Parent.Context.StartCycleCount + 1;

Invoke := THIS^;
END_METHOD

(*~
	<docu>
		<summary>
			Executes when task is aborted.
		</summary>			
	</docu>	
~*)
METHOD PROTECTED OnAbort
END_METHOD

(*~
	<docu>
		<summary>
			Executes when task reaches the ```Done``` state .
		</summary>			
	</docu>	
~*)
METHOD PROTECTED OnDone
END_METHOD

(*~
	<docu>
		<summary>
			Executes until task is in ```Error``` state .
		</summary>			
	</docu>	
~*)
METHOD PROTECTED OnTaskError
END_METHOD

(*~
	<docu>
		<summary>
			Gets whether the task is ready to be started (Tasks start by calling the <see cref="TcoTask.PlcTcoTask.Invoke()"/> method).
		</summary>			
	</docu>	
~*)
PROPERTY Ready : BOOL
GET
Ready := THIS^._taskState = eTaskState.Ready;
END_GET
END_PROPERTY

(*~
	<docu>
		<summary>
			Restores this instance to the Ready state. Can be called explicitly or from within one of the restore mechanisms.
			<para>
				See also <see cref="TcoTask.PlcTcoTask.AutoRestorable()"/>
			</para>
		</summary>			
	</docu>	
~*)
METHOD Restore : ITcoRestorable
THIS^._taskState := eTaskState.Ready;
Restore := THIS^;
END_METHOD

(*~
	<docu>
		<summary>
			Gets the actual state of this instance. 
			<para>
				See <see cref="eTaskState"/> for more details.
			</para>
		</summary>			
	</docu>	
~*)
PROPERTY State : eTaskState
GET
State := _taskState;
END_GET
END_PROPERTY

(*~
	<docu>
		<summary>
			When called with ```inCondition``` ```TRUE``` causes transition of the task into the ```Error``` state.
		</summary>			
	</docu>	
~*)
METHOD ThrowWhen
VAR_INPUT
	inCondition : BOOL;
END_VAR
IF (inCondition) THEN
	THIS^._taskState := eTaskState.Error;
END_IF
END_METHOD

END_FUNCTION_BLOCK

// POUs/MAIN
PROGRAM MAIN

END_PROGRAM

// POUs/Prototypes/TcoObject/TcoObject
(*~
	<docu>
		<summary>
			Basic construction block from which all blocks of a TcOpen application should derive in order to take advantage of the framework. 
			This function block is abstract and must be implemented in a derived block.
			```TcoObject```, must be constructed via ```FB_init(ITcoObject)``` method at instantiation. 
			```TcoObjects``` that belong to same ```TcoContext``` share the same context. 
			This is typically achieved by constructing the object with ```FB_init(THIS^)```, where ```THIS^``` is of ```ITcoObject``` (note that ITcoContext also implements ITcoObject).            			
			<para>
				<example>
				<note type="Example">
				<para>
					All the variables _myContext, _ContextTcoObjectA, _ContextTcoObjectB, _ContextChildTcoObject should have all the same value.
				</para>
				<para>
					All the variables _myIdentity, _TcoObjectAidentity, _TcoObjectBidentity, _ChildTcoObjectidentity should have uniques values.
				</para>
					<code>
							//Definition of the myTcoObject 
							FUNCTION_BLOCK myTcoObject EXTENDS TcoObject
							VAR
								  _myChildTcoObject	:	myChildTcoObject(THIS^);
							END_VAR
						
						
							//Definition of the myTcoContext 
							FUNCTION_BLOCK myTcoContext EXTENDS TcoContext
							VAR
								  _myTcoObjectA		:	myTcoObject(THIS^);					
								  _myTcoObjectB		:	myTcoObject(_myTcoObjectA.Context); 
								  _myContext		:	ITcoContext;
								  _ContextTcoObjectA	:	ITcoContext;
								  _ContextTcoObjectB	:	ITcoContext;
								  _ContextChildTcoObject	:	ITcoContext;
								  _myIdentity		:	ULINT;
								  _TcoObjectAidentity	: 	ULINT;
								  _TcoObjectBidentity	: 	ULINT;
								  _ChildTcoObjectidentity	: 	ULINT;							
							END_VAR
						
							//Plc code of the myTcoContext 
							_myContext		:= 		THIS^.Context;
							_ContextTcoObjectA	:=		_myTcoObjectA.Context;
							_ContextTcoObjectB	:=		_myTcoObjectB.Context;
							_ContextChildTcoObject	:=		_myTcoObjectB._myChildTcoObject.Context;
							_myIdentity		:=		THIS^.Identity;
							_TcoObjectAidentity	:=		_myTcoObjectA.Identity;
							_TcoObjectBidentity	:=		_myTcoObjectB.Identity;
							_ChildTcoObjectidentity	:=		_myTcoObjectB._myChildTcoObject.Identity;
					</code>
					 <note type="Explanation">
						<para>
							The context of the myTcoContext instance is assigned to itself. As the _myTcoObjectA context is assigned to this instance of the myTcoContext, it is assigned to the same context,
							and the value of the _ContextTcoObjectA will be the same as the value of the _myContext.
						</para>					
						<para>
							The context of the _myTcoObjectB instance is assigned to the _myTcoObjectA, that has already assigned context to this instance of the myTcoContext.
							So the value of the _ContextTcoObjectB will be the same as the values of the _ContextTcoObjectA and _myContext.
						</para>					
						<para>
							The context of the _myTcoObjectB._myChildTcoObject instance is assigned to the _myTcoObjectB, that has already assigned context to _myTcoObjectA, 
							that has already assigned its context to this instance of the myTcoContext.
							So the value of the _ContextChildTcoObject wile be the same as the values _ContextTcoObjectB,_ContextTcoObjectA and _myContext.
						</para>
						<para>
							As the Identities of all objects points to the themselves, all identities will have different values, as all objects are unique.
						</para>					
					 </note>
				 </note>
				</example>
			</para>
 		</summary>			
	</docu>	
~*)
FUNCTION_BLOCK ABSTRACT TcoObject IMPLEMENTS ITcoObject 
VAR
	{attribute clr [RenderIgnore()]}
	{attribute clr [ReadOnly()]}
	_Identity : ULINT;
	{attribute 'hide'}
	_Parent : ITcoObject;	
	{attribute clr [RenderIgnore()]}
	_messenger : TcoMessenger(THIS^);
END_VAR

(*~
	<docu>
		<summary>
			Gets the context of the this object. The context is provided by parent object(s).			
		</summary>			
	</docu>	
~*)
PROPERTY PUBLIC Context : ITcoContext
GET
Context := THIS^._Parent.Context;
END_GET
END_PROPERTY

(*~
	<docu>
		<summary>
			Compares this object to another object and returns ```true``` when the reference equals. 
			When overriden in derived class custom comparison of two objects of the same type can be evaluated.						
 		</summary>			
		<note>
			Default implementation compares only if two objects share the same reference. 
			If you want to compare actual values of the objects you will need to override EqualsTo method, 
			where you evaluate the values for equality.
		</note>
		<example>
			<code>
				// EqualsTo method override example of type MyObject
				METHOD PUBLIC EqualsTo : BOOL
				VAR_INPUT
					Object : ITcoObject;
				END_VAR
				
				VAR
					_object : POINTER TO MyObject;
				END_VAR
				//--------------------------------------------
				IF(__QUERYPOINTER(Object,  _object)) THEN
					EqualsTo := _object^._SomeNumber = THIS^._SomeNumber AND _object^._SomeString = THIS^._SomeString;
				END_IF;	
			</code>
		</example>
	</docu>	
~*)
METHOD PUBLIC EqualsTo : BOOL
VAR_INPUT
	Object : ITcoObject;
END_VAR
IF(Object.Identity <> 0) THEN
	EqualsTo := Object.Identity = THIS^.Identity;
END_IF
END_METHOD

METHOD FB_init : BOOL
VAR_INPUT
	bInitRetains : BOOL; // if TRUE, the retain variables are initialized (warm start / cold start)
	bInCopyCode : BOOL;  // if TRUE, the instance afterwards gets moved into the copy code (online change)
	Parent : ITcoObject;
END_VAR
_Identity := ADR(THIS^);
_Parent := Parent;
END_METHOD

(*~
	<docu>
		<summary>
			Gets the identity of this <see cref ="TcoObject.PlcTcoObject()"/>. 
			This value is assigned after download by calling the implicit method <c>FB_init()</c> and cannot be changed during runtime.
			This variable is used in the higher level applications.  
		</summary>			
	</docu>	
~*)
PROPERTY Identity : ULINT
GET
Identity := _Identity;
END_GET
END_PROPERTY

(*~
		<docu>
			<summary>
				Gets messenger of this object.
				See <see cref="TcoMessenger.PlcTcoMessenger()"/> for more details.
			</summary>			
		</docu>
~*)
PROPERTY Messenger : ITcoMessenger
GET
Messenger := THIS^._messenger;
END_GET
END_PROPERTY

END_FUNCTION_BLOCK

// POUs/Prototypes/TcoObject/ITcoObject
INTERFACE ITcoObject EXTENDS __SYSTEM.IQueryInterface

{attribute 'hide'}
PROPERTY Context : ITcoContext
GET
END_GET
END_PROPERTY

PROPERTY Identity : ULINT
GET
END_GET
END_PROPERTY

END_INTERFACE

// POUs/Prototypes/TcoContext/ITcoContext
INTERFACE ITcoContext EXTENDS ITcoObject

PROPERTY EndCycleCount : ULINT
GET
END_GET
END_PROPERTY

PROPERTY Environment : ITcoContextEnvironment
GET
END_GET
END_PROPERTY

PROPERTY Rtc : ITcoRtc
GET
END_GET
END_PROPERTY

PROPERTY StartCycleCount : ULINT
GET
END_GET
END_PROPERTY

END_INTERFACE

// POUs/Prototypes/TcoContext/ITcoContextEnvironment
INTERFACE ITcoContextEnvironment

PROPERTY Messaging : ITcoMessengerSettings
GET
END_GET
END_PROPERTY

END_INTERFACE

// POUs/Prototypes/TcoMessage/ITcoMessengerSettings
INTERFACE ITcoMessengerSettings

PROPERTY IsSuspended : BOOL
GET
END_GET
END_PROPERTY

PROPERTY MinLevel : eMessageCategory
GET
END_GET
SET
END_SET
END_PROPERTY

METHOD Resume : BOOL
VAR_INPUT
END_VAR
END_METHOD

METHOD Suspend
END_METHOD

END_INTERFACE

// POUs/Prototypes/TcoRtc/ITcoRtc
INTERFACE ITcoRtc

PROPERTY IsSynchronized : BOOL
GET
END_GET
END_PROPERTY

PROPERTY IsValid : BOOL
GET
END_GET
END_PROPERTY

METHOD NowLocal : DATE_AND_TIME
END_METHOD

METHOD NowLocalAsTIMESTRUCT : Tc2_Utilities.TIMESTRUCT
END_METHOD

METHOD NowUTC : DATE_AND_TIME
END_METHOD

METHOD NowUTCAsTIMESTRUCT : Tc2_Utilities.TIMESTRUCT
END_METHOD

METHOD TickClock : ULINT
END_METHOD

END_INTERFACE

// POUs/Prototypes/TcoMessage/TcoMessenger
(*~
		<docu>
			<summary>
				Provides mechanism for delivering static messages to the supervising applications (SCADA/HMI).	
				<remarks>			
					<note type="important">
						Each messenger has a single placeholder for the message; it stores the most important message from the last context cycle. 
						If there are more messages in a single cycle for the same messenger then less important messages are discarded and replaced by 
						the message with the category of higher severity.	
					</note>
				</remarks>			 
			</summary>			
		
		</docu>
~*)
FUNCTION_BLOCK PUBLIC TcoMessenger IMPLEMENTS ITcoMessenger
VAR			
	(*~
		<docu>
			<summary>
				Most important message of this instance of messenger; stores the most important message from the last context cycle. 
				If there are more messages in a single cycle for the same
				messenger then less important messages are discarded and replaced by the message with the category of higher severity.			 
			</summary>			
		</docu>
	~*)
	_mime : TcoMessage;
	_Parent : ITcoObject;
	_contextIdentity : ULINT;				
END_VAR

(*~
		<docu>
			<summary>
				Adds message of 'catastrophic' category to the message queue.
				Use this category when there is a situation when the device cannot continue operations due to irrecoverable failure.				 
			</summary>		
		</docu>
~*)
METHOD PUBLIC Catastrophic
VAR_INPUT
	(*~
		<docu>
			<summary>
				Arbitrary message string.			 
			</summary>			
		</docu>
	~*)
	Message : STRING(125);
END_VAR
THIS^.Post(Message, eMessageCategory.Catastrophic);
END_METHOD

(*~
		<docu>
			<summary>
				Adds message of 'critical' category to the message queue.
				Use this category when a critical error occured, that is not recoverable by the means of software (reset/restore) and a detailed inspection is required.				 
			</summary>		
		</docu>
~*)
METHOD PUBLIC Critical
VAR_INPUT
	(*~
		<docu>
			<summary>
				Arbitrary message string.			 
			</summary>			
		</docu>
	~*)
	Message : STRING(125);
END_VAR
THIS^.Post(Message, eMessageCategory.Critical);
END_METHOD

(*~
		<docu>
			<summary>
				Adds message of 'debug' category to the message queue.	
			    Use when you need to report debug information for you as programmer. 			 
			</summary>		
		</docu>
~*)
METHOD PUBLIC Debug
VAR_INPUT
	(*~
		<docu>
			<summary>
				Arbitrary message string.			 
			</summary>			
		</docu>
	~*)
	Message : STRING(125);
END_VAR
THIS^.Post(Message, eMessageCategory.Debug);
END_METHOD

(*~
		<docu>
			<summary>
				Adds message of 'error' category to the message queue.
				Use this categoty when there is a failure that cannot be immediately recovered and an intervention is needed. This is typically a situation when a device fails
				to deliver expected result. 
				Do not use this category to report information about failed process like measurement or detection.				 
			</summary>						
		</docu>
~*)
METHOD PUBLIC Error
VAR_INPUT
	(*~
		<docu>
			<summary>
				Arbitrary message string.			 
			</summary>			
		</docu>
	~*)
	Message : STRING(125);
END_VAR
THIS^.Post(Message, eMessageCategory.Error);
END_METHOD

(*~
		<docu>
			<summary>
				Adds message of 'information' category to the message queue.	
				Use when you want to deliver information to the user, that has only informative character and does not adversely affect a process.			 
			</summary>			
		</docu>
~*)
METHOD PUBLIC Info 
VAR_INPUT
	(*~
		<docu>
			<summary>
				Arbitrary message string.			 
			</summary>			
		</docu>
	~*)
	Message : STRING(125);
END_VAR
THIS^.Post(Message, eMessageCategory.Info);
END_METHOD

(*~
		<docu>
			<summary>
				Adds message of 'notification' category to the message queue.
				Use this category when you want to report a notification that may be of interest to the user, but does not adveresly affect a process.			 
			</summary>				
		</docu>
~*)
METHOD Notify 
VAR_INPUT
	(*~
		<docu>
			<summary>
				Arbitrary message string.			 
			</summary>			
		</docu>
	~*)
	Message : STRING(125);
END_VAR
THIS^.Post(Message, eMessageCategory.Notification);
END_METHOD

(*~
		<docu>
			<summary>
				Adds message of 'programming error' category to the message queue.	
				Use this category to inform about a possible programming error, defect in settings or missing information at a level of programming or system or process settings.			 
			</summary>				
		</docu>
~*)
METHOD PUBLIC Programming
VAR_INPUT
	(*~
		<docu>
			<summary>
				Arbitrary message string.			 
			</summary>			
		</docu>
	~*)
	Message : STRING(125);
END_VAR
THIS^.Post(Message, eMessageCategory.ProgrammingError);
END_METHOD

(*~
		<docu>
			<summary>
				Adds message of 'trace' category to the message queue.	
				Use when you need to track detailed information about internal states of the program for detailed visibility. 
				This is lowest level of category that can be used in production, for detailed observation of PLC program.			 
			</summary>					
		</docu>
~*)
METHOD PUBLIC Trace 
VAR_INPUT
	(*~
		<docu>
			<summary>
				Arbitrary message string.			 
			</summary>			
		</docu>
	~*)
	Message : STRING(125);
END_VAR
THIS^.Post(Message, eMessageCategory.Trace);
END_METHOD

(*~
		<docu>
			<summary>
				Adds message of 'warning' category to the message queue.
				Use this category when you want to report to the user an information about a possible problem, that may adversly affect a process.
				Information in this cateogory aims to help the user to identify a problem, the cause of such problem does not necessarily stops the process.				 
			</summary>					
		</docu>
~*)
METHOD PUBLIC Warning 
VAR_INPUT
	(*~
		<docu>
			<summary>
				Arbitrary message string.			 
			</summary>			
		</docu>
	~*)
	Message : STRING(125);
END_VAR
THIS^.Post(Message, eMessageCategory.Warning);
END_METHOD

(*~
		<docu>
			<summary>
				Clears the message content.
				<remarks>			
					<note type="important">
						This method is exposed for Rpc calls, for testing purposes. Rpc calls of this method must not be used in production code
					</note>
				</remarks>								 
			</summary>		
		</docu>
~*)
{attribute 'TcRpcEnable'}
METHOD Clear
_mime.TimeStamp :=  DT#1970-01-01-00:00;
_mime.Text := '';
_mime.Identity := 0;
_mime.Category := eMessageCategory.None;
_mime.Cycle := 0;	
_mime.PerCycleCount := 0;
END_METHOD

METHOD PROTECTED FINAL Compose 
VAR_INPUT
	Text : STRING(125);
	Category : eMessageCategory;
END_VAR
IF(_Parent <> 0 AND_THEN _Parent.Context <> 0 AND_THEN _Parent.Context.Rtc <> 0) THEN
	_mime.TimeStamp :=  _Parent.Context.Rtc.NowLocal();
	_mime.Text := Text;
	_mime.Identity := _Parent.Identity;
	_mime.Category := Category;
	_mime.Cycle := _Parent.Context.StartCycleCount;	
END_IF;
END_METHOD

METHOD FB_init : BOOL
VAR_INPUT
	bInitRetains : BOOL; // if TRUE, the retain variables are initialized (warm start / cold start)
	bInCopyCode : BOOL;  // if TRUE, the instance afterwards gets moved into the copy code (online change)
	Parent : ITcoObject;
END_VAR
_Parent := Parent;
_contextIdentity := Parent.Identity;
END_METHOD

(*~
		<docu>
			<summary>
				Creates message of given category for this messenger.				 
			</summary>				
		</docu>
~*)
METHOD PUBLIC Post 
VAR_INPUT
	(*~
		<docu>
			<summary>
				Arbitrary message string.			 
			</summary>			
		</docu>
	~*)
	Message : STRING(125);
	(*~
		<docu>
			<summary>
				Message category.			 
			</summary>			
		</docu>
	~*)
	Category : eMessageCategory;	
END_VAR
IF(_Parent <> 0 AND_THEN _Parent.Context <> 0 AND_THEN _Parent.Context.Environment <> 0 AND_THEN _Parent.Context.Environment.Messaging <> 0) THEN
	IF(Category < THIS^._Parent.Context.Environment.Messaging.MinLevel
	  OR _Parent.Context.Environment.Messaging.IsSuspended) THEN
		RETURN;
	END_IF; 	
	
	_mime.PerCycleCount := _mime.PerCycleCount + 1;
	// Same cycle filter for most important messge.
	IF(_mime.Cycle = _Parent.Context.StartCycleCount) THEN		 	
		IF(Category > _mime.Category) THEN	 
			Compose(Message, Category);
		END_IF;
	ELSE
	// Different cycle		
		_mime.PerCycleCount := 1;	
		Compose(Message, Category);		
	END_IF;	
END_IF;
END_METHOD

END_FUNCTION_BLOCK

// POUs/Prototypes/TcoMessage/ITcoMessenger
INTERFACE ITcoMessenger

(*~
		<docu>
			<summary>
				Adds message of 'debug' category to the message queue.				 
			</summary>		
		</docu>
~*)
METHOD PUBLIC Debug
VAR_INPUT
	(*~
		<docu>
			<summary>
				Arbitrary message string.			 
			</summary>			
		</docu>
	~*)
	Message : STRING(125);
END_VAR
END_METHOD

(*~
		<docu>
			<summary>
				Adds message of 'error' category to the message queue.				 
			</summary>						
		</docu>
~*)
METHOD PUBLIC Error
VAR_INPUT
	(*~
		<docu>
			<summary>
				Arbitrary message string.			 
			</summary>			
		</docu>
	~*)
	Message : STRING(125);
END_VAR
END_METHOD

(*~
		<docu>
			<summary>
				Adds message of 'information' category to the message queue.				 
			</summary>			
		</docu>
~*)
METHOD PUBLIC Info 
VAR_INPUT
	(*~
		<docu>
			<summary>
				Arbitrary message string.			 
			</summary>			
		</docu>
	~*)
	Message : STRING(125);
END_VAR
END_METHOD

(*~
		<docu>
			<summary>
				Adds message of 'notification' category to the message queue.				 
			</summary>				
		</docu>
~*)
METHOD Notify 
VAR_INPUT
	(*~
		<docu>
			<summary>
				Arbitrary message string.			 
			</summary>			
		</docu>
	~*)
	Message : STRING(125);
END_VAR
END_METHOD

(*~
		<docu>
			<summary>
				Adds message of given category to the message queue.				 
			</summary>	
			<returns>Message index.</returns>		
		</docu>
~*)
METHOD PUBLIC Post 
VAR_INPUT
	(*~
		<docu>
			<summary>
				Arbitrary message string.			 
			</summary>			
		</docu>
	~*)
	Message : STRING(125);
	(*~
		<docu>
			<summary>
				Message category.			 
			</summary>			
		</docu>
	~*)
	Category : eMessageCategory;	
END_VAR
END_METHOD

(*~
		<docu>
			<summary>
				Adds message of 'programming error' category to the message queue.				 
			</summary>				
		</docu>
~*)
METHOD PUBLIC Programming
VAR_INPUT
	(*~
		<docu>
			<summary>
				Arbitrary message string.			 
			</summary>			
		</docu>
	~*)
	Message : STRING(125);
END_VAR
END_METHOD

(*~
		<docu>
			<summary>
				Adds message of 'trace' category to the message queue.				 
			</summary>					
		</docu>
~*)
METHOD PUBLIC Trace 
VAR_INPUT
	(*~
		<docu>
			<summary>
				Arbitrary message string.			 
			</summary>			
		</docu>
	~*)
	Message : STRING(125);
END_VAR
END_METHOD

(*~
		<docu>
			<summary>
				Adds message of 'warning' category to the message queue.				 
			</summary>					
		</docu>
~*)
METHOD PUBLIC Warning 
VAR_INPUT
	(*~
		<docu>
			<summary>
				Arbitrary message string.			 
			</summary>			
		</docu>
	~*)
	Message : STRING(125);
END_VAR
END_METHOD

END_INTERFACE

// POUs/Prototypes/TcoTask/ITcoTask
INTERFACE ITcoTask EXTENDS ITcoObject, ITcoRestorable

METHOD Abort
END_METHOD

PROPERTY Busy : BOOL
GET
END_GET
END_PROPERTY

PROPERTY Done : BOOL
GET
END_GET
END_PROPERTY

PROPERTY Error : BOOL
GET
END_GET
END_PROPERTY

(*~
	<docu>
		<summary>
			Use to start the execution of the task. The starting is possible from Ready state.
			<para>Moreover it is also possible to start the task again from Done state by performing the '''rising edge''' of the calling of the Invoke() method.</para>
			<p>Analogously to the xExecute signal of the <a href="https://plcopen.org/sites/default/files/downloads/creating_plcopen_compliant_function_block_libraries.pdf" title="Title"> PLCopen </a> motion function blocks.</p>			
		</summary>			
	</docu>	
~*)
METHOD Invoke : ITcoTaskStatus
END_METHOD

END_INTERFACE

// POUs/Prototypes/TcoRestorable/ITcoRestorable
INTERFACE ITcoRestorable EXTENDS __SYSTEM.IQueryInterface

METHOD Restore : ITcoRestorable
END_METHOD

END_INTERFACE

// POUs/Prototypes/TcoTask/ITcoTaskStatus
INTERFACE ITcoTaskStatus

PROPERTY Busy : BOOL
GET
END_GET
END_PROPERTY

PROPERTY Done : BOOL
GET
END_GET
END_PROPERTY

PROPERTY Error : BOOL
GET
END_GET
END_PROPERTY

END_INTERFACE

// POUs/Prototypes/TcoState/TcoState
FUNCTION_BLOCK TcoState EXTENDS TcoStateBase

METHOD PUBLIC ChangeState : ITcoState
VAR_INPUT
	NewState : INT;
END_VAR
ChangeState := SUPER^.ChangeStateProtected(NewState);
END_METHOD

END_FUNCTION_BLOCK

// POUs/Prototypes/TcoState/TcoStateBase
(*~
	<docu>
		<summary>
			Provides basic state controller. It could be implemented using <c>IF</c>, <c>IF</c> <c>ELSIF</c> or <c>CASE</c> statement. The transition to the different state needs to be perfromed by calling 
			<see cref="TcoState.PlcTcoState.ChangeState(Object)"/> method. This method ensures also calling the <see cref="TcoState.PlcTcoState.OnStateChange(Object,Object)"/> every time that state is changed. The 
		  	<c>OnStateChange()</c>could be overloaded and some custom code that needs to be executed on each change of the state could be placed here. The TcoState could be used like this:
			<para>
				<example>
				<note type="Example 1">
				<para>
					<c>_myTask()</c> is not a member of this <c>TcoState()</c>, it is restored manually to be able to trigger it in the next state.
				</para>
					<code>
						IF State = 10 THEN
							Main._myTask.Invoke();
							Main._myTask.Execute();
							IF Main._myTask.Done THEN
								ChangeState(State + 10);
								Main._myTask.Restore();
							END_IF
						END_IF
						IF State = 20 THEN
							Main._myTask.Invoke();
							Main._myTask.Execute();
							IF Main._myTask.Done THEN
								ChangeState(State + 10);
								Main._myTask.Restore();
							END_IF
						END_IF
					</code>
				 </note>
				</example>
			</para>		
			<para>
				<example>
				<note type="Example 2">
				<para>
					<c>_myTask()</c> is a member of this <c>TcoState()</c>, it is restored manually using the fluent syntax to be able to trigger it in the next state.
				</para>
					<code>
						CASE State OF
							10:	
							_myTask.Invoke();
							_myTask.Execute();
							IF _myTask.Done THEN
								ChangeState(State + 10).RestoreObject(_myTask);
							END_IF
							20:
							_myTask.Invoke();
							_myTask.Execute();
							IF _myTask.Done THEN
								ChangeState(State + 10).RestoreObject(_myTask);
							END_IF	
						END_CASE
					</code>
				 </note>
				</example>
				<para>
					See <see cref="TcoState.PlcTcoState.RestoreObject(Object)"/> for more details.
				</para>
			</para>			
		</summary>		
	</docu>	
~*)	
FUNCTION_BLOCK ABSTRACT TcoStateBase EXTENDS TcoObject IMPLEMENTS ITcoState, ITcoObjectRestorer
VAR
	{attribute clr [ReadOnly()]}
	_State : INT; 	
	{attribute 'hide'}
	_enableAutoRestore : BOOL;
	{attribute 'hide'}
	_AutoRestorable : BOOL;
	{attribute 'hide'}
	_StartCycleCount	: ULINT;
	{attribute 'hide'}
	_MyParentsChangeStateCycle	: ULINT;
	{attribute 'hide'}
	_ChangeStateCycle	: ULINT;
	{attribute 'hide'}
	_LastChangedState	: INT;
	{attribute 'hide'}
	_MyParentsLastChangedState	: INT;	
END_VAR

(*~
	<docu>
		<summary>
			Returns if this instance is auto restorable. This is 'dependency property'. Value of this property is given by the parent of this object. 
			This value is assigned after download by calling the implicit method <c>FB_init()</c> of the parent object and cannot be changed during runtime.
			The <c>AutoRestorable</c> property of this objects is retrieved from the <c>EnableAutoRestore</c> property of the parent object.
			This is done by calling the <c>CheckIfAutoRestoreEnabledByParent()</c> method inside the implicit method <c>FB_init()</c> after download.
			If this instance is the auto restorable it will call the <see cref="TcoState.PlcTcoState.Restore()"/> method if:
			<para>
				1.) This instance has not been called for one or more cycles and starts to be called again. (By calling the instance means asking for its property <see cref="TcoState.PlcTcoState.State()"/> property).
			</para>
			<para>
				2.)	Parent object of this instance changes its state.
			</para>
			<para>
				See also <see cref="TcoState.PlcTcoState.EnableAutoRestore()"/>
			</para>
		</summary>			
	</docu>	
~*)
PROPERTY AutoRestorable : BOOL
GET
AutoRestorable := _AutoRestorable;
END_GET
END_PROPERTY

(*~
	<docu>
		<summary>
			Private method called each time that State property is asked for. If this instance is auto restorable, this method ensures calling the <see cref="TcoState.PlcTcoState.Restore()"/> method if:
			<para>
				1.)	Parent object of this instance changes its state in this Plc cycle.
			</para>
			<para>
				2.)	Parent object of this instance changes its state no mather when and this instance has not yet process this change.
			</para>
			<para>
				3.) This instance has not been called for one or more cycles and starts to be called again. (By calling the instance means asking for its property <see cref="TcoState.PlcTcoState.State()"/> property).
			</para>
			<para>
				See also <see cref="TcoState.PlcTcoState.AutoRestorable()"/>
			</para>
			<para>
				See also <see cref="TcoState.PlcTcoState.EnableAutoRestore()"/>
			</para>
		</summary>			
	</docu>	
~*)
METHOD PRIVATE AutoRestore
VAR 
	_MyParent_TcoState	: ITcoState := 0;
	_MyParent_ChangeStateCycle : ULINT;
	_MyParent_LastChangeState : INT;
END_VAR
//If parent of this instance is TcoState type or its derived type and the parent
//EnableAutoRestore property is set to TRUE, this instance determines the value
//of its own AutoRestorable property by calling CheckIfAutoRestoreEnabledByParent 
//after each download.
IF _AutoRestorable THEN		
	IF __QUERYINTERFACE(THIS^._Parent,_MyParent_TcoState) THEN 
		_MyParent_ChangeStateCycle := _MyParent_TcoState.LastStateChangeCycle;
		_MyParent_LastChangeState := _MyParent_TcoState.State;
	END_IF;	
	//If OnStateChange event of the parent has occured, the value of the parent's 
	//StartCycleCount property is stored into its ChangeStateCycle property.
	//Each child has to deal with it individually in the next call of its body,
	//restore itself, and copy the parent's ChangeStateCycle property into the
	//child's own property.
	IF _MyParent_ChangeStateCycle <> _MyParentsChangeStateCycle THEN
		THIS^.Restore();
		_MyParentsChangeStateCycle := _MyParent_ChangeStateCycle;
	END_IF
	IF _MyParent_LastChangeState <> _MyParentsLastChangedState THEN
		THIS^.Restore();
		_MyParentsLastChangedState := _MyParent_LastChangeState;
	END_IF
END_IF
END_METHOD

(*~
	<docu>
		<summary>
			Use to change the State property of this instance to the new value. This method is final, so it cannot be overloaded. However there is a <see cref="TcoState.PlcTcoState.OnStateChange(Object,Object)"/> 
			method that is called on each change of the <c>State</c> and could be overloaded.
			<para>
				<example>
				<note type="Example">
				<para>
					Possibility to use the fluent syntax.
				</para>
					<code>ChangeState(newState).RestoreObject(myChildObject);</code>
				 </note>
				</example>
			</para>		
		</summary>			
	</docu>	
~*)
METHOD PROTECTED ChangeStateProtected : ITcoState 
VAR_INPUT
	NewState : INT;
END_VAR
VAR 
	PreviousState	: INT;
END_VAR
PreviousState := THIS^._State;
THIS^._State := NewState;

IF NewState <> PreviousState THEN
	_ChangeStateCycle := THIS^.Context.StartCycleCount;
	_LastChangedState  := NewState;
	OnStateChange(PreviousState,NewState);
END_IF;

ChangeStateProtected := THIS^;
END_METHOD

(*~
	<docu>
		<summary>
			This method ensures reading out the parent's <see cref="TcoState.PlcTcoState.EnableAutoRestore()/> property and writing it into the <see cref="TcoState.PlcTcoState.AutoRestorable()"/> of this instance.
			Calling this method is ensured by calling the implicit method <c>FB_init()</c> after download, or after online change.
		</summary>			
	</docu>	
~*)
{attribute 'call_after_online_change_slot' := '100'}
METHOD PRIVATE CheckIfAutoRestoreEnabledByParent
VAR
	_MyParent_TcoState	: 	ITcoState := 0;
END_VAR
IF __QUERYINTERFACE(THIS^._Parent,_MyParent_TcoState) THEN 
	_AutoRestorable := _MyParent_TcoState.IsAutoRestoreEnabled;
END_IF;
END_METHOD

(*~
	<docu>
		<summary>
			Private method called each time that the <see cref="TcoState.PlcTcoState.State()"/> property is asked for. 
			If this instance is auto restorable, this method ensures calling the <see cref="TcoState.PlcTcoState.Restore()"/> method if
			this instance has not been called for one or more cycles and starts to be called again. (By calling the instance means asking for its property State).
			<para>
				See also <see cref="TcoState.PlcTcoState.AutoRestorable()"/>
			</para>
			<para>
				See also <see cref="TcoState.PlcTcoState.EnableAutoRestore()"/>
			</para>
		</summary>			
	</docu>	
~*)
METHOD PRIVATE CheckIfCalledCyclically
VAR 
	_MyContextStartCycleCount : ULINT;
END_VAR
//If parent of this instance is TcoState type or its derived type and the parent
//EnableAutoRestore property is set to TRUE, this instance determines the value
//of its own AutoRestorable property by calling CheckIfAutoRestoreEnabledByParent 
//after each download.
IF _AutoRestorable THEN		
	_MyContextStartCycleCount := THIS^.Context.StartCycleCount;
	//If this instance is AutoRestorable, its body has to be called cyclically, 
	//otherwise this instance is restored.
	//This mechanism force the user to call this instance properly,
	//in order to don't miss the OnStateChange() event of the parent
	//in case of the body of this instance isn't called.
	IF _MyContextStartCycleCount > _StartCycleCount + 1 THEN
		THIS^.Restore();
	END_IF
	_StartCycleCount := _MyContextStartCycleCount;
END_IF
END_METHOD

(*~
	<docu>
		<summary>
			Returns the context of the parent object, that this object is assigned to.
			This context is given by declaration, its value is assigned after download by calling the implicit method <c>FB_init()</c> and cannot be changed during runtime.
		</summary>			
	</docu>	
~*)
PROPERTY Context : ITcoContext
GET
Context := THIS^._Parent.Context;
END_GET
END_PROPERTY

METHOD FB_init : BOOL
VAR_INPUT
	bInitRetains : BOOL; // if TRUE, the retain variables are initialized (warm start / cold start)
	bInCopyCode : BOOL;  // if TRUE, the instance afterwards gets moved into the copy code (online change)
	Parent : ITcoObject;
	AutoRestoreMode : eRestoreMode; 
END_VAR
_Identity 		:=	ADR(THIS^);
_Parent			:=	Parent;
_enableAutoRestore	:=	AutoRestoreMode = eRestoreMode.AutoRestoreMembers;

CheckIfAutoRestoreEnabledByParent();
END_METHOD

(*~
	<docu>
		<summary>
			Returns the own identity of the <see cref ="TcoState.PlcTcoState()"/>. This value is assigned after download by calling the implicit method <c>FB_init()</c> and cannot be changed during runtime.
			This variable is used in the higher level packages.  
		</summary>			
	</docu>	
~*)
PROPERTY Identity : ULINT
GET
Identity := _Identity;
END_GET
END_PROPERTY

(*~
	<docu>
		<summary>
			Returns if the auto restore mechanism is enabled for this instance. This property does not affect this instance, but it affects all members of this instance.
			If the auto restore is enabled, the child member call its <c>Restore()</c> method if:
			<para>
			1.) Its instance has not been called for one or more cycles.
			</para>
			<para>
			2.)	Its parent object (THIS^ instance) has changed its state.
			</para>
			This value is assigned after download by calling the implicit method <c>FB_init()</c> and cannot be changed during runtime.
			<para>
				See also <see cref="TcoState.PlcTcoState.AutoRestorable()"/>
			</para>
		</summary>			
	</docu>	
~*)
PROPERTY IsAutoRestoreEnabled : BOOL
GET
IsAutoRestoreEnabled := _enableAutoRestore;
END_GET
END_PROPERTY

(*~
	<docu>
		<summary>
			Returns number of the Plc cycle during which this instance changes its <c>State</c> last time.
			The child objects ask for this value to ensure auto restore mechanism working.  	
		</summary>			
	</docu>	
~*)
PROPERTY LastStateChangeCycle : ULINT
GET
LastStateChangeCycle := _ChangeStateCycle;
END_GET
END_PROPERTY

(*~
	<docu>
		<summary>
			This method is called on each change of the <c>State</c>. This method could be overloaded and custom code should be placed here.	
		</summary>			
	</docu>	
~*)
METHOD PROTECTED OnStateChange
VAR_INPUT
	PreviousState	: INT;
	NewState 		: INT;
END_VAR
END_METHOD

(*~
	<docu>
		<summary>
			Restore this instance to the state -1. Could be called explicitly so as using auto restore mechanism.
			<para>
				<example>
					<note type="Example">
						<para>
							Possibility to use the fluent syntax.
						</para>
						<code>
							Restore().RestoreObject(myFirstChildObject).RestoreObject(mySecondChildObject);
						</code>
					 </note>
				</example>
			</para>				
			<para>
				See also <see cref="TcoState.PlcTcoState.AutoRestorable()"/>
			</para>
			<para>
				See also <see cref="TcoState.PlcTcoState.EnableAutoRestore()"/>
			</para>
		</summary>			
	</docu>	
~*)
METHOD Restore : ITcoRestorable
ChangeStateProtected(-1);

Restore := THIS^;
END_METHOD

(*~
	<docu>
		<summary>
			Ensures calling the <c>Restore()</c> method on the object entered.	
			<para>
				<example>
				<note type="Example">
				<para>
					Possibility to use the fluent syntax.
				</para>
					<code>ChangeState(newState).RestoreObject(myFirstChildObject).RestoreObject(mySecondChildObject);</code>
				 </note>
				</example>
			</para>		
		</summary>			
	</docu>	
~*)
METHOD RestoreObject : ITcoObjectRestorer
VAR_INPUT
	Obj : ITcoRestorable;
END_VAR
Obj.Restore();
RestoreObject := THIS^;
END_METHOD

(*~
	<docu>
		<summary>
			Return actual state of this instance. Needs to be asked for cyclically in case of this instance is auto restorable.
			<para>
				See also <see cref="TcoState.PlcTcoState.AutoRestorable()"/>
			</para>
		</summary>			
	</docu>	
~*)
PROPERTY State : INT
GET
CheckIfCalledCyclically();
AutoRestore();

State := _State;
END_GET
END_PROPERTY

END_FUNCTION_BLOCK

// POUs/Prototypes/TcoState/ITcoState
INTERFACE ITcoState EXTENDS ITcoObject, ITcoRestorable

PROPERTY IsAutoRestoreEnabled : BOOL
GET
END_GET
END_PROPERTY

PROPERTY LastStateChangeCycle : ULINT
GET
END_GET
END_PROPERTY

METHOD RestoreObject : ITcoObjectRestorer
VAR_INPUT
	Obj : ITcoRestorable;
END_VAR
END_METHOD

PROPERTY State : INT
GET
END_GET
END_PROPERTY

END_INTERFACE

// POUs/Prototypes/TcoRestorable/ITcoObjectRestorer
INTERFACE ITcoObjectRestorer

(*~
	<docu>
		<summary>
			Ensures calling the <c>Restore()</c> method on the object entered.	
			<para>
				<example>
				<note type="Example">
				<para>
					Possibility to use the fluent syntax.
				</para>
					<code>ChangeState(newState).RestoreObject(myFirstChildObject).RestoreObject(mySecondChildObject);</code>
				 </note>
				</example>
			</para>		
		</summary>			
	</docu>	
~*)
METHOD RestoreObject : ITcoObjectRestorer
VAR_INPUT
	Obj : ITcoRestorable;
END_VAR
END_METHOD

END_INTERFACE

// POUs/Prototypes/TcoComponent/ITcoServiceable
INTERFACE ITcoServiceable

PROPERTY IsService : BOOL
GET
END_GET
END_PROPERTY

METHOD PUBLIC Service
END_METHOD

END_INTERFACE

// POUs/Prototypes/TcoRtc/TcoRtc
FUNCTION_BLOCK PUBLIC TcoRtc IMPLEMENTS ITcoRtc
VAR
	{attribute 'hide'}
	_isValid							:	BOOL := FALSE;
	{attribute 'hide'}
	_state								:	UINT;
	{attribute 'hide'}
	_TimeZoneID							:	Tc2_Utilities.E_TimeZoneID;
	{attribute 'hide'}
	_NT_GetLocalTime					: 	Tc2_Utilities.NT_GetTime;
	{attribute 'hide'}
	_FB_TzSpecificLocalTimeToSystemTime :	Tc2_Utilities.FB_TzSpecificLocalTimeToSystemTime;
	{attribute 'hide'}
	_RTC_EX2							:	RTC_EX2;
	{attribute 'hide'}
	_PDT	 							:	Tc2_Utilities.TIMESTRUCT;	
	{attribute 'hide'}
	_LocalTime 							:	Tc2_Utilities.TIMESTRUCT;
	{attribute clr [ReadOnly()]}
	_LocalTimeDT						:	DATE_AND_TIME;
	{attribute 'hide'}
	_UTCTime 							:	Tc2_Utilities.TIMESTRUCT;
	{attribute clr [ReadOnly()]}
	_UTCTimeDT							:	DATE_AND_TIME;
END_VAR

PROPERTY IsSynchronized : BOOL
GET
IsSynchronized :=  RtcPrg._isSynchronized;
END_GET
END_PROPERTY

PROPERTY IsValid : BOOL
GET
IsValid := _isValid;
END_GET
END_PROPERTY

METHOD NowLocal : DATE_AND_TIME
IF _isValid THEN
	NowLocal := _LocalTimeDT;
END_IF
END_METHOD

METHOD NowLocalAsTIMESTRUCT : Tc2_Utilities.TIMESTRUCT
IF _isValid THEN
	NowLocalAsTIMESTRUCT := _LocalTime;
END_IF
END_METHOD

METHOD NowUTC : DATE_AND_TIME
IF _isValid THEN
	NowUTC := _UTCTimeDT;
END_IF
END_METHOD

METHOD NowUTCAsTIMESTRUCT : Tc2_Utilities.TIMESTRUCT
IF _isValid THEN
	NowUTCAsTIMESTRUCT := _UTCTime;
END_IF
END_METHOD

METHOD TickClock : ULINT
TickClock := Tc2_EtherCAT.F_GetActualDcTime64();
END_METHOD

METHOD INTERNAL Update
IF _state = 0 THEN
	_isValid := FALSE;
	_NT_GetLocalTime(NETID := '127.0.0.1.1.1', START := TRUE);
	IF _NT_GetLocalTime.BUSY AND NOT _NT_GetLocalTime.ERR THEN 
		_state := _state + 10;
	END_IF
END_IF
	
IF _state = 10 THEN
	_NT_GetLocalTime(START := FALSE);
	IF NOT _NT_GetLocalTime.BUSY AND NOT _NT_GetLocalTime.ERR THEN 
		_state := _state + 10;
	END_IF
END_IF

IF _state = 20 THEN
	_NT_GetLocalTime(START := FALSE);
		
	_PDT := _NT_GetLocalTime.TIMESTR;

	_isValid := TRUE;
//	_state := 0;
END_IF

_RTC_EX2(EN := _isValid, PDT := _PDT);

_LocalTime := _RTC_EX2.CDT;
_LocalTimeDT := Tc2_Utilities.SYSTEMTIME_TO_DT(_LocalTime);

IF RtcPrg._isSynchronized THEN
	_FB_TzSpecificLocalTimeToSystemTime(in 		:=	_LocalTime,
										tzInfo 	:=	RtcPrg._TimeZoneInformation,
										out		=>	_UTCTime,
										eTzID	=>	_TimeZoneID);

	_UTCTimeDT := Tc2_Utilities.SYSTEMTIME_TO_DT(_UTCTime);
END_IF
END_METHOD

END_FUNCTION_BLOCK

// POUs/Prototypes/TcoRtc/RtcPrg
PROGRAM INTERNAL RtcPrg
VAR
	{attribute 'hide'}
	_RtcSynchParams						:	RtcSynchParams;			
	{attribute 'hide'}
	_isSynchronized						:	BOOL := FALSE;
	{attribute 'hide'}
	_state								:	UINT;
	{attribute 'hide'}
	_syncAmsIdIsLocale					:	BOOL;
	{attribute 'hide'}
	_FB_GetLocalAmsNetId 				: 	Tc2_Utilities.FB_GetLocalAmsNetId;
	{attribute 'hide'}
	_FB_GetTimeZoneInformation			:	Tc2_Utilities.FB_GetTimeZoneInformation;
	{attribute 'hide'}
	_FB_SetTimeZoneInformation			:	Tc2_Utilities.FB_SetTimeZoneInformation;
	{attribute 'hide'}
	_TimeZoneInformation				:	Tc2_Utilities.ST_TimeZoneInformation;
	{attribute 'hide'}
	_TimeZoneID							:	Tc2_Utilities.E_TimeZoneID;
	{attribute 'hide'}
	_startTime							:	Tc2_EtherCAT.T_DCTIME64;
	{attribute 'hide'}
	_endTime							:	Tc2_EtherCAT.T_DCTIME64;
	{attribute 'hide'}
	_getOffset							:	Tc2_EtherCAT.T_DCTIME64;
	{attribute 'hide'}
	_setOffset							:	Tc2_EtherCAT.T_DCTIME64;
	{attribute 'hide'}
	_NT_GetSyncTime						: 	Tc2_Utilities.NT_GetTime;
	{attribute 'hide'}
	_NT_SetLocalTime 					: 	Tc2_Utilities.NT_SetLocalTime;
	{attribute 'hide'}
	_NT_GetLocalTime					: 	Tc2_Utilities.NT_GetTime;
	{attribute 'hide'}
	_FB_TzSpecificLocalTimeToSystemTime :	Tc2_Utilities.FB_TzSpecificLocalTimeToSystemTime;
	{attribute 'hide'}
	_remote2localDiff					:	Tc2_EtherCAT.T_DCTIME64;
	{attribute 'hide'}
	_offset								:	ULINT;
	{attribute 'hide'}
	_syncCounter						:	ULINT;
	{attribute 'hide'}
	_lastSyncTick						: 	Tc2_EtherCAT.T_DCTIME64;
	{attribute 'hide'}
	_timeTick							: 	Tc2_EtherCAT.T_DCTIME64;
	{attribute 'hide'}
	_LocalTime 							:	Tc2_Utilities.TIMESTRUCT;
	{attribute 'hide'}
	_UTCTime 							:	Tc2_Utilities.TIMESTRUCT;
END_VAR

METHOD INTERNAL Synchronize
VAR_INPUT
	inRtcSynchParams	: RtcSynchParams;
END_VAR
IF _RtcSynchParams.synchContextIdentity = 0 AND inRtcSynchParams.synchContextIdentity <> 0 THEN
	_RtcSynchParams.synchContextIdentity := inRtcSynchParams.synchContextIdentity;
END_IF

IF _RtcSynchParams.synchContextIdentity <>0 AND _RtcSynchParams.synchContextIdentity = inRtcSynchParams.synchContextIdentity THEN
	_RtcSynchParams.doSynch := inRtcSynchParams.doSynch;
	_RtcSynchParams.syncAmsId := inRtcSynchParams.syncAmsId;
	_RtcSynchParams.syncPeriod := inRtcSynchParams.syncPeriod;
	IF _NT_GetLocalTime.ERR THEN
		_NT_GetLocalTime(START := FALSE);
		_isSynchronized := FALSE;
		RETURN;	
	END_IF

	IF _state = 0 THEN
		IF _RtcSynchParams.doSynch THEN
			_isSynchronized := FALSE;
			_state := _state + 10;
		ELSE 
			_isSynchronized := FALSE;
			_state := 210;
		END_IF
	END_IF
	
	IF _state = 10 THEN
		_FB_GetLocalAmsNetId(bExecute := TRUE);
		IF _FB_GetLocalAmsNetId.bBusy AND NOT _FB_GetLocalAmsNetId.bError THEN
			_state := _state + 10;
		END_IF
	END_IF
	
	IF _state = 20 THEN
		_FB_GetLocalAmsNetId(bExecute := FALSE);
		IF NOT _FB_GetLocalAmsNetId.bBusy AND NOT _FB_GetLocalAmsNetId.bError THEN
			_state := _state + 10;
		END_IF
	
	END_IF
	
	IF _state = 30 THEN
		_syncAmsIdIsLocale := 	_RtcSynchParams.syncAmsId = _FB_GetLocalAmsNetId.AddrString OR 
								_RtcSynchParams.syncAmsId = '127.0.0.1.1.1' OR 
								_RtcSynchParams.syncAmsId = '';
		_state := _state + 10;
	END_IF
	
	IF _state = 40 THEN
		_startTime := Tc2_EtherCAT.F_GetActualDcTime64();
		_state := _state + 10;
	END_IF
	
	IF _state = 50 THEN
		_FB_GetTimeZoneInformation(sNetID := _RtcSynchParams.syncAmsId, bExecute := TRUE);
		IF _FB_GetTimeZoneInformation.bBusy AND NOT _FB_GetTimeZoneInformation.bError THEN
			_state := _state + 10;
		END_IF
	END_IF
	
	IF _state = 60 THEN
		_FB_GetTimeZoneInformation(bExecute := FALSE);
		IF NOT _FB_GetTimeZoneInformation.bBusy AND NOT _FB_GetTimeZoneInformation.bError THEN
			_state := _state + 10;
		END_IF
	END_IF
	
	IF _state = 70 THEN
		_TimeZoneInformation := _FB_GetTimeZoneInformation.tzInfo;
		_TimeZoneID := _FB_GetTimeZoneInformation.tzID;
		_endTime := Tc2_EtherCAT.F_GetActualDcTime64();
		_getOffset := (_endTime - _startTime ) / 2;
		_state := _state + 10;
	END_IF
	
	IF _state = 80 THEN
		IF _syncAmsIdIsLocale THEN
			_state := 180;
		ELSE
			_state := _state + 10;
		END_IF
	END_IF
	
	IF _state = 90 THEN
		_startTime := Tc2_EtherCAT.F_GetActualDcTime64();
		_state := _state + 10;
	END_IF
	
	IF _state = 100 THEN
		_FB_SetTimeZoneInformation(sNetID := '127.0.0.1.1.1', tzInfo := _TimeZoneInformation , bExecute := TRUE);
		IF _FB_SetTimeZoneInformation.bBusy AND NOT _FB_SetTimeZoneInformation.bError THEN
			_state := _state + 10;
		END_IF
	END_IF
	
	IF _state = 110 THEN
		_FB_SetTimeZoneInformation(bExecute := FALSE);
		IF NOT _FB_SetTimeZoneInformation.bBusy AND NOT _FB_SetTimeZoneInformation.bError THEN
			_state := _state + 10;
		END_IF
	END_IF
	
	IF _state = 120 THEN
		_endTime := Tc2_EtherCAT.F_GetActualDcTime64();
		_setOffset := (_endTime - _startTime ) / 2;
		_state := _state + 10;
	END_IF
	
	IF _state = 130 THEN
		_NT_GetSyncTime(NETID := _RtcSynchParams.syncAmsId, START := TRUE);
		IF _NT_GetSyncTime.BUSY AND NOT _NT_GetSyncTime.ERR THEN 
			_state := _state + 10;
		END_IF
	END_IF
	
	IF _state = 140 THEN
		_NT_GetSyncTime(START := FALSE);
		IF NOT _NT_GetSyncTime.BUSY AND NOT _NT_GetSyncTime.ERR THEN
			_state := _state + 10;
		END_IF
	END_IF
	
	IF _state = 150 THEN
		_NT_GetSyncTime(START := FALSE);
		_offset := LREAL_TO_ULINT(ULINT_TO_LREAL(_getOffset + _setOffset) / 1000000) * 1000000;
		_offset := _offset + Tc2_EtherCAT.SYSTEMTIME_TO_DCTIME64(_NT_GetSyncTime.TIMESTR,0,0) + _getOffset + _setOffset;	
		_LocalTime := Tc2_EtherCAT.DCTIME64_TO_SYSTEMTIME(_offset);
		_state := _state + 10;
	END_IF
	
	IF _state = 160 THEN
		_NT_GetSyncTime(START := FALSE);
		_NT_SetLocalTime(	NETID := '127.0.0.1.1.1', 
							TIMESTR := _LocalTime,
							START := TRUE);
		IF _NT_SetLocalTime.BUSY AND NOT _NT_SetLocalTime.ERR THEN 
			_state := _state + 10;
		END_IF
	END_IF
	
	IF _state = 170 THEN
		_NT_GetSyncTime(START := FALSE);
		_NT_SetLocalTime(START := FALSE);
		IF NOT _NT_SetLocalTime.BUSY AND NOT _NT_SetLocalTime.ERR THEN
			_state := _state + 10;
		END_IF
	END_IF
	
	IF _state = 180 THEN
		_NT_GetSyncTime(NETID := _RtcSynchParams.syncAmsId, START := TRUE);
		_NT_GetLocalTime(NETID := '127.0.0.1.1.1', START := TRUE);
		IF _NT_GetSyncTime.BUSY AND NOT _NT_GetSyncTime.ERR AND NOT _NT_GetLocalTime.ERR THEN 
			_state := _state + 10;
		END_IF
	END_IF
	
	IF _state = 190 THEN
		_NT_GetSyncTime(START := FALSE);
		_NT_GetLocalTime(START := FALSE);
		IF NOT _NT_GetSyncTime.BUSY AND NOT _NT_GetSyncTime.ERR AND NOT _NT_GetLocalTime.BUSY AND NOT _NT_GetLocalTime.ERR THEN 
			_state := _state + 10;
		END_IF
	END_IF
	
	IF _state = 200 THEN
		_remote2localDiff := Tc2_EtherCAT.SYSTEMTIME_TO_DCTIME64(_NT_GetSyncTime.TIMESTR,0,0) -  Tc2_EtherCAT.SYSTEMTIME_TO_DCTIME64(_NT_GetLocalTime.TIMESTR,0,0);
	
		_NT_GetSyncTime(START := FALSE);
		_NT_GetLocalTime(START := FALSE);
		_NT_SetLocalTime(START := FALSE);
	
		_LocalTime := _NT_GetLocalTime.TIMESTR;
		_FB_TzSpecificLocalTimeToSystemTime(in 		:=	_LocalTime,
											tzInfo 	:=	_TimeZoneInformation,
											out		=>	_UTCTime,
											eTzID	=>	_TimeZoneID);
	
		_lastSyncTick := Tc2_EtherCAT.F_GetActualDcTime64(); 	
	
		_syncCounter := _syncCounter + 1;
		_state := _state + 10;
	END_IF
	
	IF _state = 210 THEN
		_NT_GetLocalTime(NETID := '127.0.0.1.1.1', START := TRUE);
		IF _NT_GetLocalTime.BUSY AND NOT _NT_GetLocalTime.ERR THEN 
			_state := _state + 10;
		END_IF
	END_IF
	
	IF _state = 220 THEN
		_NT_GetLocalTime(START := FALSE);
		IF NOT _NT_GetLocalTime.BUSY AND NOT _NT_GetLocalTime.ERR THEN 
			_state := _state + 10;
		END_IF
	END_IF
	
	IF _state = 230 THEN
		_isSynchronized := TRUE;
		_NT_GetSyncTime(START := FALSE);
		_NT_GetLocalTime(START := FALSE);
		_NT_SetLocalTime(START := FALSE);
		
		_timeTick :=Tc2_EtherCAT.F_GetActualDcTime64(); 	
		
		IF _RtcSynchParams.doSynch THEN
			IF (_timeTick - _lastSyncTick) / 1000000000  >= _RtcSynchParams.syncPeriod THEN
				_state := 0;
			ELSE
				_state := 210;
			END_IF
		ELSE
			_state := 210;
		END_IF
	END_IF
END_IF
END_METHOD

END_PROGRAM

// POUs/Prototypes/TcoContext/TcoContextEnvironment
FUNCTION_BLOCK TcoContextEnvironment IMPLEMENTS ITcoContextEnvironment
VAR
	_messenger : TcoMessengerSettings;
END_VAR

(*~
		<docu>
			<summary>
				Gets messaging settings of this context.			
			</summary>			
		</docu>	
~*)
PROPERTY Messaging : ITcoMessengerSettings
GET
Messaging := _messenger;
END_GET
END_PROPERTY

END_FUNCTION_BLOCK

// POUs/Prototypes/TcoMessage/TcoMessengerSettings
FUNCTION_BLOCK INTERNAL TcoMessengerSettings IMPLEMENTS ITcoMessengerSettings
VAR
	_minLevel : eMessageCategory;
	_isMessagingSuspended : BOOL;	
END_VAR

(*~
	<docu>
		<summary>
			Gets whether the messaging is suspended at this point in program.					
			<para>
				See also <see cref="TcoMessengerSettings.Resume()"/>
			</para>
			<para>
				See also <see cref="TcoMessengerSettings.Suspend()"/>
			</para>
			<para>
				See also <see cref="TcoMessengerSettings.MinLevel"/>
			</para>
		</summary>			
	</docu>	
~*)
PROPERTY PUBLIC IsSuspended : BOOL
GET
IsSuspended := _isMessagingSuspended;
END_GET
END_PROPERTY

(*~
	<docu>
		<summary>
			Gets or set minimal messaging level, the objects will post only messages for the levels of this or superior severity.					
			<para>
				See also <see cref="TcoMessengerSettings.Resume()"/>
			</para>
			<para>
				See also <see cref="TcoMessengerSettings.Suspend()"/>
			</para>
			<para>
				See also <see cref="TcoMessengerSettings.MinLevel"/>
			</para>
		</summary>			
	</docu>	
~*)
PROPERTY PUBLIC MinLevel : eMessageCategory
GET
MinLevel := _minLevel;
END_GET
SET
_minLevel := MinLevel;
END_SET
END_PROPERTY

(*~
	<docu>
		<summary>
			Resumes messaging from the all objects of this context, when the messaging was previously suspended by ```Suspend``` method.					
			<para>
				See also <see cref="TcoMessengerSettings.Suspend()"/>
			</para>
			<para>
				See also <see cref="TcoMessengerSettings.MinLevel"/>
			</para>
		</summary>			
	</docu>	
~*)
METHOD PUBLIC Resume : BOOL
_isMessagingSuspended := FALSE;
END_METHOD

(*~
	<docu>
		<summary>
			Suspends messaging from the all objects of this context that would occur from this point in the call tree.						
			<para>
				See also <see cref="TcoMessengerSettings.Resume()"/>
			</para>
			<para>
				See also <see cref="TcoMessengerSettings.MinLevel"/>
			</para>
		</summary>			
	</docu>	
~*)
METHOD PUBLIC Suspend
_isMessagingSuspended := TRUE;
END_METHOD

END_FUNCTION_BLOCK

// POUs/Compatibility/TcoContextNfCompatibility
FUNCTION_BLOCK FINAL TcoContextNfCompatibility EXTENDS TcoContextCompatibility

METHOD PROTECTED FINAL Main
END_METHOD

METHOD PUBLIC VolatileClose
THIS^._Close();
END_METHOD

METHOD PUBLIC VolatileOpen
THIS^._Open();
END_METHOD

END_FUNCTION_BLOCK

// POUs/Prototypes/TcoComponent/ITcoComponent
INTERFACE ITcoComponent EXTENDS ITcoObject,ITcoRestorable, ITcoServiceable

END_INTERFACE

// POUs/Prototypes/TcoComponent/TcoComponent
(*~
	<docu>
		<summary>
			Basic class for components.
		</summary>				
	</docu>	
~*)
FUNCTION_BLOCK ABSTRACT TcoComponent EXTENDS TcoObject IMPLEMENTS ITcoComponent
VAR
	{attribute 'hide'}
	_serviceContexCycle : ULINT;	
(*~
	<docu>
		<summary>
			True if component is in service mode.
		</summary>			
	</docu>	
~*)
	{attribute addProperty Name "<#In service mode#>"}
	{attribute clr [ReadOnly()]}
	_inServiceMode : BOOL;	
END_VAR

CheckIfIsInServiceMode();

METHOD INTERNAL CheckIfIsInServiceMode 
VAR
	_myContextCycleCount : ULINT;
END_VAR
_myContextCycleCount := Context.StartCycleCount;
//When component.Service() is called "before" invoking its task _serviceContexCycle is equal to Context.StartCycleCount
//When component.Service() is called "after" invoking its task (_serviceContexCycle + 1) is equal to Context.StartCycleCount
//otherwise _serviceContexCycle should be lower then Context.StartCycleCount until Context.StartCycleCount overflow its range
//which should occur cca every 585 mil years at 1ms PLC task.    
_inServiceMode := _serviceContexCycle = _myContextCycleCount OR (_serviceContexCycle + 1) = _myContextCycleCount;
END_METHOD

METHOD FB_init : BOOL
VAR_INPUT
	bInitRetains : BOOL; // if TRUE, the retain variables are initialized (warm start / cold start)
	bInCopyCode : BOOL;  // if TRUE, the instance afterwards gets moved into the copy code (online change)
	Parent : ITcoObject;
END_VAR
SUPER^.FB_init(bInitRetains, bInCopyCode, Parent);
END_METHOD

(*~
	<docu>
		<summary>
			Gets whether the component is in serviceable state. Serviceable state is when ```Service``` method is called cyclicaly.   
		</summary>			
	</docu>	
~*)
PROPERTY IsService : BOOL
GET
CheckIfIsInServiceMode();
IsService := _inServiceMode;
END_GET
END_PROPERTY

(*~
	<docu>
		<summary>
			Restores this instance to the Ready state. Can be called explicitly or from within one of the restore mechanisms.	
		</summary>			
	</docu>	
~*)
METHOD ABSTRACT Restore : ITcoRestorable
END_METHOD

(*~
	<docu>
		<summary>
			Executes the logic for manual-maintenance control.   
		</summary>			
	</docu>	
~*)
METHOD PUBLIC FINAL Service
_serviceContexCycle := Context.StartCycleCount;
ServiceMode();
END_METHOD

(*~
	<docu>
		<summary>
		    Custom service (manual, maintenance) logic.
			This method must be implemented in derived class.
		</summary>			
	</docu>	
~*)
METHOD PROTECTED ABSTRACT ServiceMode
END_METHOD

END_FUNCTION_BLOCK

// POUs/Prototypes/TcoSequencer/ITcoSequencer
INTERFACE ITcoSequencer EXTENDS ITcoState

(*~
	<docu>
		<summary>
			Gets the information about the current step.						
		</summary>				
	</docu>	
~*)
PROPERTY CurrentStep : REFERENCE TO StepDetails
GET
END_GET
END_PROPERTY

PROPERTY ModeController : ITcoSequencerModeController
GET
END_GET
END_PROPERTY

(*~
	<docu>
		<summary>
			<para>
				Ensures calling the Open(), Main() and Close() methods in the desired order.
				This method is final, so it cannot be overloaded. The InstanceName.Run() needs to be called cyclically inside the appropriate context.
			</para>
		</summary>			
	</docu>	
~*)
METHOD PUBLIC FINAL Run
END_METHOD

END_INTERFACE

// POUs/Prototypes/TcoSequencer/ITcoSequencerModeController
INTERFACE ITcoSequencerModeController

(*~
	<docu>
		<summary>			
			Gets or sets sequencer mode.
			<remarks>			
				<para>
					See <see cref="eSequencerMode"/> for detailed description.
				</para>
			</remarks>		
		</summary>			
	</docu>	
~*)
PROPERTY PUBLIC Mode : eSequencerMode
GET
END_GET
SET
END_SET
END_PROPERTY

(*~
	<docu>
		<summary>
			This method triggers StepBackward task, that decrements current step (variable: <c> TcoSequencer._theOrderOfTheCurrentlyExecutedStep</c> ), in case the sequencer is in step mode, and the current step is greather than zero.
		</summary>			
	</docu>	
~*)
METHOD PUBLIC FINAL StepBackward
END_METHOD

(*~
	<docu>
		<summary>
			This method triggers StepForward task, that increment current step (variable: <c>TcoSequencer._theOrderOfTheCurrentlyExecutedStep</c> ), 
			in case the sequencer is in step mode, and the current step is lower than number of steps in th sequence (variable: <c>TcoSequencer._numberOfStepsInSequence</c> ).
		</summary>			
	</docu>	
~*)
METHOD PUBLIC FINAL StepForward
END_METHOD

(*~
	<docu>
		<summary>
			Triggers StepIn task, that changes the current step status from ReadyToRun to Running. 
			This causes starting the execution of the body of the current step.
		</summary>			
	</docu>	
~*)
METHOD PUBLIC FINAL StepIn
END_METHOD

END_INTERFACE

// POUs/Prototypes/TcoSequencer/TcoSequencer
(*~
		<docu>
			<summary>
				Provides basic sequential control, including step mode, which allows to run the sequence step-by-step, steping forward and steping backward.
			</summary>
		</docu>		
~*)
FUNCTION_BLOCK ABSTRACT TcoSequencer EXTENDS TcoStateExtendible IMPLEMENTS ITcoSequencer
VAR CONSTANT 
    MinStepID : INT := -32768;
    MaxStepID : INT := 32767;
END_VAR 
VAR
(*~
	<docu>
		<summary>
			Holds the status information about current step.
		</summary>			
		<remarks>			
			<para>
				See <see cref="StepDetails"/> for detailed description.
			</para>
		</remarks>		
	</docu>	
~*)
	{attribute addProperty Name "<#Current step#>"}
	_currentStep : StepDetails;
(*~
	<docu>
		<summary>
			True if an error occurs in the sequence. Detailed cause of this error is described by the _sequencerErrorId.		
		</summary>				
		<remarks>			
			<para>
				See <see cref="TcoSequencer.PlcTcoSequencer._sequencerErrorId"/> for detailed description.
			</para>
		</remarks>	
	</docu>	
~*)	
	{attribute addProperty Name "<#Sequencer error#>"}
	{attribute clr [ReadOnly()]}
	_sequencerHasError : BOOL;
(*~
	<docu>
		<summary>
			Describes cause of the sequencer error.
		</summary>		
		<remarks>			
			<para>
				See <see cref="eSequencerError"/> for detailed description.
			</para>
		</remarks>			
	</docu>	
~*)	
	{attribute addProperty Name "<#Sequencer error ID#>"}
	{attribute clr [ReadOnly()]}
	_sequencerErrorId : eSequencerError := eSequencerError.noError;
(*~
	<docu>
		<summary>
			Handles changing the sequencer mode (Cyclic, Step).
		</summary>		
	</docu>	
~*)	
	_modeController : TcoSequencerModeController(THIS^);
(*~
	<docu>
		<summary>
			Elapsed time of presently running sequence cycle.
		</summary>		
	</docu>	
~*)	
	{attribute addProperty Name "<#Sequence cycle elapsed time#>"}	
	_SequenceElapsedTime : TIME;
(*~
	<docu>
		<summary>
			Elapsed time of the currently executing step.
		</summary>		
	</docu>	
~*)	
	{attribute addProperty Name "<Current step time#>"}	
	_StepElapsedTime : TIME;
(*~
	<docu>
		<summary>
			Total time of the last sequence cycle. 
		</summary>		
	</docu>	
~*)	
	{attribute addProperty Name "<#Total sequence time#>"}	
	_LastCycleTime: TIME;
END_VAR
VAR
	{attribute 'hide'}
	_isFirstStepEntry : BOOL;
	{attribute 'hide'}
	_theOrderOfTheCurrentlyEvaluatedStep : UINT;	
	{attribute 'hide'}
	_theOrderOfTheCurrentlyExecutedStep : UINT;	
	{attribute 'hide'}
	_theOrderOfThePreviouslyExecutedStep : UINT;
	 {attribute 'hide'}
	_IdOfThePreviouslyExecutedStep : INT;
	{attribute 'hide'}
	_numberOfStepsInSequence : UINT;
	{attribute 'hide'}
	_previousNumberOfStepsInSequence : UINT;
	{attribute 'hide'}
	_stepCounter : UINT;	
	{attribute 'hide'}
	_requestStepActive : BOOL;	
	{attribute 'hide'}
	_requestedStepId : INT := MinStepID;	
	{attribute 'hide'}
	_cycleTimer : TON;   
	{attribute 'hide'}
	_StepTimer : TON;
	{attribute 'hide'}
	_requestStepCycle: UINT;
	{attribute 'hide'}
	_StepIdChanged : BOOL;
	{attribute 'hide'}
	_StepOrderChanged : BOOL;
	{attribute 'hide'}
	_ChangeStepIdFrom : INT;
	{attribute 'hide'}
	_ChangeStepIdTo : INT;
	{attribute 'hide'}
	_ChangeStepOrderFrom : UINT;
	{attribute 'hide'}
	_ChangeStepOrderTo : UINT;
	{attribute 'hide'}
	_stepIdUniquenessChecked : BOOL := FALSE;
	{attribute 'hide'}
	_checkStepIdRequestedInStepMode : BOOL;
	{attribute 'hide'}
	_restoringSequence : BOOL;	
END_VAR

VAR
	{attribute 'hide'}
    _pPreviusSteps : POINTER TO INT;
END_VAR

VAR
	_lastActiveCycle : ULINT;
END_VAR

(*~
	<docu>
		<summary>
			Performs the check of the ```StepId``` of the currently executed step.
			<remarks>			
				<note type="important">
					The StepId of each step in the sequence must be unique throughout the complete sequence, and it must not be changed.
					```StepId``` sould be assigned as a number literal or a constant.
				</note>
			</remarks>			
		</summary>			
	</docu>	
~*)
METHOD PRIVATE CheckStepId : BOOL
VAR_INPUT
	inStepID : INT;
	inStepModeActive : BOOL;
	inStepInRunning : BOOL;	
END_VAR
CheckStepID := TRUE;

IF((_IdOfThePreviouslyExecutedStep <> inStepID) AND NOT _isFirstStepEntry AND (NOT inStepModeActive OR inStepInRunning)) THEN
	IF (_theOrderOfTheCurrentlyExecutedStep =0) AND (_theOrderOfTheCurrentlyEvaluatedStep = 0) AND (_IdOfThePreviouslyExecutedStep =0) THEN
		_IdOfThePreviouslyExecutedStep := inStepID;
	ELSIF NOT _StepIdChanged AND NOT _StepOrderChanged THEN	 
		_StepIdChanged := TRUE;
		_ChangeStepIdFrom := _IdOfThePreviouslyExecutedStep;
		_ChangeStepIdTo := inStepID;
		CheckStepID := FALSE;
	END_IF;		
END_IF
END_METHOD

(*~
	<docu>
		<summary>
			Implicit call of this method is ensured by calling the method Run().
			It must not be called explicitely by consumer code in derived blocks.
			<remarks>			
				<note type="important">
					Do not call this method explicitly.
				</note>
			</remarks>
		</summary>			
	</docu>	
~*)
METHOD INTERNAL FINAL Close
_previousNumberOfStepsInSequence := _numberOfStepsInSequence;

IF _modeController._stepIn.Done THEN
	_modeController._stepIn.Restore();	
END_IF

_restoringSequence := FALSE;
END_METHOD

(*~
	<docu>
		<summary>
			<para>
				Completes the sequencer, and return the sequencer pointer to the first step in the seuqence.
				Method is typically called inside the last step of the sequence.
			</para>
		</summary>			
	</docu>	
~*)
METHOD PROTECTED FINAL CompleteSequence
_theOrderOfTheCurrentlyExecutedStep := 0;
_LastCycleTime := _SequenceElapsedTime;
_cycleTimer(IN:= FALSE, PT:= T#0S);	

_currentStep.Status := eStepStatus.Done;

OnSequenceCompleted();

_modeController._stepForward.Restore();
_modeController._stepBackward.Restore();
_modeController._stepIn.Restore();
END_METHOD

